(* IEC 61131-3 sources: GHEP-MITSU_BACKUP/, 12 files *)

(* ---- encoder_speed_calc.st ---- *)
(* ============================================================================ *)
(* PROGRAM: POU_ENCODER_SPEED (Fixed Scan 10ms - Ngắt chu kỳ 10ms)             *)
(* MACHINE: MÁY GHÉP MÀNG METALIZE                                             *)
(* HARDWARE: 03 Module QD62 tại Slot 1 (H20), Slot 2 (H30), Slot 3 (H40)        *)
(* ENCODERS: 5 Trục (T = Thu, X1 = Xả 1, X2 = Master, M = Metalize, S = Dầu)     *)
(* ============================================================================ *)

VAR_GLOBAL
    (* --- DỮ LIỆU TỐC ĐỘ ĐỌC VỀ VÀ TÍNH TOÁN (HMI / PROGRAM DÙNG CHUNG) --- *)
    (* Tốc độ vòng/phút (RPM x10: 1500 -> 150.0 RPM) *)
    RPM_T       : DINT := 0; (* Trục Thu T *)
    RPM_X1      : DINT := 0; (* Trục Xả X1 *)
    RPM_X2      : DINT := 0; (* Trục Master X2 *)
    RPM_M       : DINT := 0; (* Trục Metalize M *)
    RPM_S       : DINT := 0; (* Trục Dầu S *)

    (* Tốc độ dây mét/phút (MPM x10: 1205 -> 120.5 MPM) *)
    MPM_T       : DINT := 0; (* Vận tốc dây Trục Thu T *)
    MPM_X1      : DINT := 0; (* Vận tốc dây Trục Xả X1 *)
    MPM_X2      : DINT := 0; (* Vận tốc dây Trục Master X2 (Tốc độ chuẩn dòng máy) *)
    MPM_M       : DINT := 0; (* Vận tốc dây Trục Metalize M *)
    MPM_S       : DINT := 0; (* Vận tốc dây Trục Dầu S *)

    (* Cài đặt đường kính lô (mm) *)
    Dia_T_mm    : DINT := 150; (* Đường kính cuộn Thu T *)
    Dia_X1_mm   : DINT := 150; (* Đường kính cuộn Xả X1 *)
    Dia_X2_mm   : DINT := 200; (* Đường kính lô Master X2 (Cố định 200mm) *)
    Dia_M_mm    : DINT := 180; (* Đường kính lô Metalize M *)
    Dia_S_mm    : DINT := 160; (* Đường kính lô Dầu S *)

    (* Cài đặt độ phân giải Encoder PPR (xung/vòng) *)
    PPR_Encoder : DINT := 2000; (* 2000 PPR x 4 = 8000 pulses/rev *)

    (* Biến lưu xung vòng trước *)
    Prev_Pulse_T  : DINT := 0;
    Prev_Pulse_X1 : DINT := 0;
    Prev_Pulse_X2 : DINT := 0;
    Prev_Pulse_M  : DINT := 0;
    Prev_Pulse_S  : DINT := 0;
END_VAR

VAR
    (* Biến xung hiện tại đọc từ Buffer Memory QD62 *)
    Curr_Pulse_T  : DINT := 0;
    Curr_Pulse_X1 : DINT := 0;
    Curr_Pulse_X2 : DINT := 0;
    Curr_Pulse_M  : DINT := 0;
    Curr_Pulse_S  : DINT := 0;

    (* Delta xung đếm được trong 10ms *)
    Delta_T  : DINT := 0;
    Delta_X1 : DINT := 0;
    Delta_X2 : DINT := 0;
    Delta_M  : DINT := 0;
    Delta_S  : DINT := 0;

    (* PPR tổng sau khi nhân 4 pha A/B *)
    Total_PPR : DINT := 8000;
END_VAR

(* ============================================================================ *)
(* MAIN BODY: CHẠY TRONG POU CHU KỲ NGẮT FIXED SCAN 10MS                      *)
(* ============================================================================ *)

(* --- 1. KÍCH HOẠT CỜ CHO PHÉP ĐẾM XUNG CHO 3 MODULE QD62 --- *)
Y21 := TRUE; (* QD62 #1 (Slot 1 H20) CH1: Enable Trục Thu T *)
Y22 := TRUE; (* QD62 #1 (Slot 1 H20) CH2: Enable Trục Xả X1 *)

Y31 := TRUE; (* QD62 #2 (Slot 2 H30) CH1: Enable Trục Master X2 *)
Y32 := TRUE; (* QD62 #2 (Slot 2 H30) CH2: Enable Trục Metalize M *)

Y41 := TRUE; (* QD62 #3 (Slot 3 H40) CH1: Enable Trục Dầu S *)

(* --- 2. ĐỌC XUNG 32-BIT TỪ BUFFER MEMORY G2/G3 VÀ G10/G11 --- *)
(* QD62 #1 (Slot 1 - H20) *)
DMOV(TRUE, U1\G2,  Curr_Pulse_T);  (* CH1: Trục Thu T *)
DMOV(TRUE, U1\G10, Curr_Pulse_X1); (* CH2: Trục Xả X1 *)

(* QD62 #2 (Slot 2 - H30) *)
DMOV(TRUE, U2\G2,  Curr_Pulse_X2); (* CH1: Trục Master X2 *)
DMOV(TRUE, U2\G10, Curr_Pulse_M);  (* CH2: Trục Metalize M *)

(* QD62 #3 (Slot 3 - H40) *)
DMOV(TRUE, U3\G2,  Curr_Pulse_S);  (* CH1: Trục Dầu S *)

(* --- 3. TÍNH DELTA XUNG NỐI TIẾP TRONG 10MS (100Hz) --- *)
Delta_T  := ABS(Curr_Pulse_T  - Prev_Pulse_T);
Delta_X1 := ABS(Curr_Pulse_X1 - Prev_Pulse_X1);
Delta_X2 := ABS(Curr_Pulse_X2 - Prev_Pulse_X2);
Delta_M  := ABS(Curr_Pulse_M  - Prev_Pulse_M);
Delta_S  := ABS(Curr_Pulse_S  - Prev_Pulse_S);

(* Cập nhật xung vòng trước *)
Prev_Pulse_T  := Curr_Pulse_T;
Prev_Pulse_X1 := Curr_Pulse_X1;
Prev_Pulse_X2 := Curr_Pulse_X2;
Prev_Pulse_M  := Curr_Pulse_M;
Prev_Pulse_S  := Curr_Pulse_S;

Total_PPR := PPR_Encoder * 4; (* Nhân 4 độ phân giải mode 2-Phase 4x *)

(* --- 4. TÍNH TỐC ĐỘ VÒNG/PHÚT RPM (RPM x10: 1500 -> 150.0 RPM) --- *)
(* Công thức: RPM = (Delta_Pulse * 60000ms / 10ms) / Total_PPR *)
IF Total_PPR > 0 THEN
    RPM_T  := (Delta_T  * 600000) / Total_PPR;
    RPM_X1 := (Delta_X1 * 600000) / Total_PPR;
    RPM_X2 := (Delta_X2 * 600000) / Total_PPR;
    RPM_M  := (Delta_M  * 600000) / Total_PPR;
    RPM_S  := (Delta_S  * 600000) / Total_PPR;
END_IF;

(* --- 5. TÍNH VẬN TỐC DÂY MÉT/PHÚT MPM (MPM x10: 1205 -> 120.5 MPM) --- *)
(* Công thức: MPM = (RPM * PI * Dia_mm) / 1000 *)
(* PI x 1000 = 3142 *)
MPM_T  := (RPM_T  * 3142 * Dia_T_mm)  / 1000000;
MPM_X1 := (RPM_X1 * 3142 * Dia_X1_mm) / 1000000;
MPM_X2 := (RPM_X2 * 3142 * Dia_X2_mm) / 1000000; (* Vận tốc Master dây chuyền *)
MPM_M  := (RPM_M  * 3142 * Dia_M_mm)  / 1000000;
MPM_S  := (RPM_S  * 3142 * Dia_S_mm)  / 1000000;

(* ---- metalize_main_program.st ---- *)
(* ============================================================================ *)
(* MAIN PROGRAM: POU_MAIN_METALIZE (BỔ SUNG CHỐNG TRÙNG MÀNG & CHỐNG KHÔ KEO/DẦU S, Ms) *)
(* PLC: Q02UCPU | Base Rack Slot 0..6                                           *)
(* CỜ M130/M131: BẬT/TẮT TORQUE HÃM M & U KHI DỪNG MÁY CHỐNG TRÙNG MÀNG          *)
(* CỜ M132/M133: QUAY BÒ CHẬM TRỤC S & TRỤC Ms KHI DỪNG MÁY CHỐNG KHÔ KEO/DẦU  *)
(* ============================================================================ *)

VAR_GLOBAL
    (* --- BẢNG ĐIỀU KHIỂN HMI WEINTEK --- *)
    HMI_Auto_Mode       : BOOL := TRUE;
    HMI_Reset_Error     : BOOL := FALSE;
    HMI_Start           : BOOL := FALSE;
    HMI_Stop            : BOOL := FALSE;
    HMI_Inc_Hold        : BOOL := FALSE;
    HMI_Dec_Hold        : BOOL := FALSE;
    HMI_PID_Enable      : BOOL := TRUE;

    (* --- CỜ CHỐNG TRÙNG MÀNG KHI DỪNG MÁY (HOLD TORQUE WHEN STOPPED) --- *)
    Hold_Torque_Stop_M  : BOOL := TRUE;  (* ON: Giữ Torque Thắng M khi dừng chống trùng màng *)
    Hold_Torque_Stop_U  : BOOL := TRUE;  (* ON: Giữ Torque Xả U khi dừng chống trùng màng *)

    (* --- CỜ QUAY BÒ CHẬM CHỐNG KHÔ KEO / DẦU CHO TRỤC S & Ms KHI DỪNG MÁY --- *)
    Anti_Dry_Rotate_S   : BOOL := TRUE;  (* ON: Cho Trục Dầu S quay bò chậm khi dừng máy *)
    Anti_Dry_Rotate_Ms  : BOOL := TRUE;  (* ON: Cho Trục Ghép Ms quay bò chậm khi dừng máy *)
    Anti_Dry_Crawl_Speed: DINT := 10;    (* Tốc độ bò chậm chống khô keo (1.0 m/phút) *)

    (* --- LỆNH BEN NÂNG/HẠ CUỘN MÀNG --- *)
    Lift_Up_T           : BOOL := FALSE;
    Lift_Down_T         : BOOL := FALSE;
    Lift_Up_M           : BOOL := FALSE;
    Lift_Down_M         : BOOL := FALSE;
    Lift_Up_U           : BOOL := FALSE;
    Lift_Down_U         : BOOL := FALSE;

    (* --- ĐIỀU KHIỂN 2 PEN ÉP MÀNG QY40 (Y66, Y67) VÀ NÚT BẤM QX40 (X52, X53) --- *)
    Release_Pen_Speed_MPM: DINT := 20;   (* Tốc độ cài đặt nhả 2 pen khi dừng máy (2.0 m/phút) *)
    Pen1_Cmd            : BOOL := FALSE; (* Trạng thái ON/OFF Pen 1 (Y66) *)
    Pen2_Cmd            : BOOL := FALSE; (* Trạng thái ON/OFF Pen 2 (Y67) *)

    (* --- CÀI ĐẶT TORQUE HÃM MIN / MAX --- *)
    Min_Torque_M        : DINT := 400;
    Max_Torque_M        : DINT := 2000;
    Init_Holding_Torque_M : DINT := 800;

    Min_Torque_U        : DINT := 500;
    Max_Torque_U        : DINT := 2500;
    Init_Holding_Torque_U : DINT := 1000;

    (* --- ĐƯỜNG KÍNH LÕI CORE DIA VÀ MAX DIA (MM) --- *)
    Core_Dia_T_mm       : DINT := 76;
    Core_Dia_M_mm       : DINT := 76;
    Core_Dia_U_mm       : DINT := 76;

    Max_Dia_T_mm        : DINT := 1000;
    Max_Dia_M_mm        : DINT := 600;
    Max_Dia_U_mm        : DINT := 800;

    (* --- TỈ LỆ TỐC ĐỘ VÀ BÙ TỐC TRỤC S --- *)
    Speed_Ratio_S       : DINT := 1000;
    Speed_Offset_S      : DINT := 0;

    (* --- TỐC ĐỘ CÀI ĐẶT DÂY CHUYỀN --- *)
    Max_Speed_MPM       : DINT := 1000;
    Min_Speed_MPM       : DINT := 20;
    Current_Line_MPM    : DINT := 0;
    Target_Line_MPM     : DINT := 0;

    (* --- TỶ SỐ TRUYỀN GEAR RATIO --- *)
    Gear_Ratio_T        : DINT := 10100;
    Gear_Ratio_X1       : DINT := 8000;
    Gear_Ratio_X2       : DINT := 8000;
    Gear_Ratio_Ms       : DINT := 10000;
    Gear_Ratio_S        : DINT := 10000;
    Gear_Ratio_U        : DINT := 1000;

    (* --- ĐƯỜNG KÍNH LÔ CƠ CẤU (MM x10) --- *)
    Dia_X1_Roller_mm    : DINT := 3005;
    Dia_X2_Roller_mm    : DINT := 3005;
    Dia_Ms_Roller_mm    : DINT := 2000;
    Dia_S_Roller_mm     : DINT := 1000;

    (* --- ĐƯỜNG KÍNH THỰC TẾ ĐÃ ĐƯỢC LỌC THÔNG THẤP (MM) --- *)
    Real_Dia_T_mm       : DINT := 76;
    Real_Dia_M_mm       : DINT := 600;
    Real_Dia_U_mm       : DINT := 800;

    (* --- ĐỘ DÀY MÀNG (MICRON) --- *)
    Thick_Paper_U_um    : DINT := 60;
    Thick_Metalize_M_um : DINT := 20;

    (* --- MÉT HÀNG ĐÃ GHÉP VÀ MÉT CÀI ĐẶT TỰ DỪNG --- *)
    Set_Target_Length   : DINT := 1000;
    Total_Length_Meters : DINT := 0;
    HMI_Reset_Length    : BOOL := FALSE;
    HMI_Reset_Roll_M    : BOOL := FALSE;
    HMI_Reset_Roll_U    : BOOL := FALSE;
    HMI_Reset_Roll_T    : BOOL := FALSE;

    (* --- LỰC CĂNG SP VÀ CALIB --- *)
    SP_Tension_T        : DINT := 1500;
    SP_Tension_X1       : DINT := 1200;
    SP_Tension_M        : DINT := 1000;
    SP_Tension_U        : DINT := 1000;

    Kp_T : DINT := 150; Ki_T : DINT := 20; Kd_T : DINT := 10;
    Kp_X1: DINT := 120; Ki_X1: DINT := 15; Kd_X1: DINT := 8;
    Kp_M : DINT := 100; Ki_M : DINT := 10; Kd_M : DINT := 5;
    Kp_U : DINT := 100; Ki_U : DINT := 10; Kd_U : DINT := 5;

    Zero_Set_T          : BOOL := FALSE;
    Zero_Set_X1         : BOOL := FALSE;
    Zero_Set_M          : BOOL := FALSE;
    Zero_Set_U          : BOOL := FALSE;

    Calib_Gain_T        : DINT := 1000;
    Calib_Gain_X1       : DINT := 1000;
    Calib_Gain_M        : DINT := 1000;
    Calib_Gain_U        : DINT := 1000;
END_VAR

VAR
    State_Machine       : INT := 0;
    Tension_Stable      : BOOL := FALSE;
    Stable_Timer        : INT := 0;
    Stop_Delay_Timer    : INT := 0;

    Trig_X50            : BOOL := FALSE;
    Trig_X51            : BOOL := FALSE;
    Mem_X50             : BOOL := FALSE;
    Mem_X51             : BOOL := FALSE;

    Trig_X52            : BOOL := FALSE; (* Sườn nút bấm Pen 1 X52 *)
    Mem_X52             : BOOL := FALSE;
    Trig_X53            : BOOL := FALSE; (* Sườn nút bấm Pen 2 X53 *)
    Mem_X53             : BOOL := FALSE;

    Curr_Pulse_X2       : DINT := 0;
    Prev_Pulse_X2       : DINT := 0;
    Accum_Pulse_X2      : DINT := 0;

    Curr_Pulse_T        : DINT := 0;
    Prev_Pulse_T        : DINT := 0;
    Accum_Pulse_T       : DINT := 0;
    Rev_Count_T         : DINT := 0;
    Rev_Count_M         : DINT := 0;
    Rev_Count_U         : DINT := 0;

    (* BIẾN LƯU XUNG ĐỂ TÍNH ĐƯỜNG KÍNH THEO TỶ SỐ XUNG KHI MÁY CHẠY (KHÔNG DÙNG ĐỘ DÀY) *)
    Last_Pulse_X2_M     : DINT := 0;
    Last_Pulse_X2_U     : DINT := 0;
    Last_Pulse_X2_T     : DINT := 0;
    Last_Pulse_T        : DINT := 0;
    Delta_Pulse_M       : DINT := 0;
    Delta_Pulse_U       : DINT := 0;
    Delta_Pulse_T_Master: DINT := 0;

    Raw_Dia_M_mm        : DINT := 600;
    Raw_Dia_U_mm        : DINT := 800;
    Raw_Dia_T_mm        : DINT := 76;

    Calc_Speed_T        : DINT := 0;
    Calc_Speed_X1       : DINT := 0;
    Calc_Speed_X2       : DINT := 0;
    Calc_Speed_Ms       : DINT := 0;
    Calc_Torque_M       : DINT := 0;
    Calc_Speed_S        : DINT := 0;
    Calc_Speed_U        : DINT := 0;

    Base_Torque_M       : DINT := 0;

    pid_T               : FB_TENSION_PID;
    pid_X1              : FB_TENSION_PID;
    pid_M               : FB_TENSION_PID;
    pid_U               : FB_TENSION_PID;

    fbCCLink            : FFB_METALIZE_CONTROL;
END_VAR

(* ============================================================================ *)
(* MAIN LOGIC                                                                   *)
(* ============================================================================ *)

(* 1. ĐIỀU KHIỂN BEN NÂNG / HẠ CUỘN MÀNG T, M, U (QY40P SLOT 5 Y60..Y65) *)
Y60 := Lift_Up_T   AND NOT(Lift_Down_T);
Y61 := Lift_Down_T AND NOT(Lift_Up_T);

Y62 := Lift_Up_M   AND NOT(Lift_Down_M);
Y63 := Lift_Down_M AND NOT(Lift_Up_M);

Y64 := Lift_Up_U   AND NOT(Lift_Down_U);
Y65 := Lift_Down_U AND NOT(Lift_Up_U);

(* 1.1 ĐIỀU KHIỂN 2 PEN ÉP MÀNG QY40 (Y66, Y67) BẰNG 2 NÚT BẤM TOGGLE QX40 (X52, X53) *)
(* Bắt sườn lên sút nhấn X52 (Pen 1) và X53 (Pen 2) trên QX40 *)
Trig_X52 := X52 AND NOT(Mem_X52);
Mem_X52  := X52;

Trig_X53 := X53 AND NOT(Mem_X53);
Mem_X53  := X53;

(* Khi bấm nút X52: Đảo trạng thái Pen 1 (ON -> OFF / OFF -> ON) *)
IF Trig_X52 THEN
    Pen1_Cmd := NOT Pen1_Cmd;
END_IF;

(* Khi bấm nút X53: Đảo trạng thái Pen 2 (ON -> OFF / OFF -> ON) *)
IF Trig_X53 THEN
    Pen2_Cmd := NOT Pen2_Cmd;
END_IF;

(* TỰ ĐỘNG NHẢ 2 PEN KHI MÁY DỪNG ĐẾN TỐC ĐỘ CÀI ĐẶT (Release_Pen_Speed_MPM) *)
(* Khi dừng máy (State 3 Stopping hoặc State 0 Stopped) và tốc độ giảm xuống <= tốc độ cài đặt *)
IF (State_Machine = 3 OR State_Machine = 0) AND (Current_Line_MPM <= Release_Pen_Speed_MPM) THEN
    Pen1_Cmd := FALSE;
    Pen2_Cmd := FALSE;
END_IF;

(* Xuất ngõ ra QY40 *)
Y66 := Pen1_Cmd; (* Ngõ ra Pen 1 trên QY40 *)
Y67 := Pen2_Cmd; (* Ngõ ra Pen 2 trên QY40 *)

(* 2. BẮT SƯỜN LÊN CẢM BIẾN TIỆM CẬN ĐO VÒNG QUAY QX40 *)
Trig_X50 := X50 AND NOT(Mem_X50); (* X50: Cuộn Metalize M *)
Mem_X50  := X50;

Trig_X51 := X51 AND NOT(Mem_X51); (* X51: Cuộn Xả Giấy U *)
Mem_X51  := X51;

(* 3. TÍNH ĐƯỜNG KÍNH THỰC TẾ KHÔNG DÙNG ĐỘ DÀY CHO CUỘN METALIZE M (QX40 X50) *)
IF HMI_Reset_Roll_M THEN
    Rev_Count_M        := 0;
    Raw_Dia_M_mm       := Max_Dia_M_mm;
    Real_Dia_M_mm      := Max_Dia_M_mm;
    Last_Pulse_X2_M    := Curr_Pulse_X2;
    HMI_Reset_Roll_M   := FALSE;
ELSIF Trig_X50 THEN
    Rev_Count_M := Rev_Count_M + 1;
    Delta_Pulse_M := Curr_Pulse_X2 - Last_Pulse_X2_M;
    Last_Pulse_X2_M := Curr_Pulse_X2;

    IF Delta_Pulse_M > 0 THEN
        (* Công thức tỷ số xung Master X2 trong 1 vòng quay cuộn M *)
        Raw_Dia_M_mm := (Delta_Pulse_M * Dia_X2_Roller_mm) / 320000;
        IF Raw_Dia_M_mm < Core_Dia_M_mm THEN Raw_Dia_M_mm := Core_Dia_M_mm; END_IF;
        IF Raw_Dia_M_mm > Max_Dia_M_mm THEN Raw_Dia_M_mm := Max_Dia_M_mm; END_IF;
    END_IF;

    IF Rev_Count_M >= 3 THEN
        Real_Dia_M_mm := Real_Dia_M_mm + ((Raw_Dia_M_mm - Real_Dia_M_mm) / 5);
    ELSE
        Real_Dia_M_mm := Max_Dia_M_mm;
    END_IF;
END_IF;

(* 4. TÍNH ĐƯỜNG KÍNH THỰC TẾ KHÔNG DÙNG ĐỘ DÀY CHO CUỘN XẢ GIẤY U (QX40 X51) *)
IF HMI_Reset_Roll_U THEN
    Rev_Count_U        := 0;
    Raw_Dia_U_mm       := Max_Dia_U_mm;
    Real_Dia_U_mm      := Max_Dia_U_mm;
    Last_Pulse_X2_U    := Curr_Pulse_X2;
    HMI_Reset_Roll_U   := FALSE;
ELSIF Trig_X51 THEN
    Rev_Count_U := Rev_Count_U + 1;
    Delta_Pulse_U := Curr_Pulse_X2 - Last_Pulse_X2_U;
    Last_Pulse_X2_U := Curr_Pulse_X2;

    IF Delta_Pulse_U > 0 THEN
        (* Công thức tỷ số xung Master X2 trong 1 vòng quay cuộn U *)
        Raw_Dia_U_mm := (Delta_Pulse_U * Dia_X2_Roller_mm) / 320000;
        IF Raw_Dia_U_mm < Core_Dia_U_mm THEN Raw_Dia_U_mm := Core_Dia_U_mm; END_IF;
        IF Raw_Dia_U_mm > Max_Dia_U_mm THEN Raw_Dia_U_mm := Max_Dia_U_mm; END_IF;
    END_IF;

    IF Rev_Count_U >= 3 THEN
        Real_Dia_U_mm := Real_Dia_U_mm + ((Raw_Dia_U_mm - Real_Dia_U_mm) / 5);
    ELSE
        Real_Dia_U_mm := Max_Dia_U_mm;
    END_IF;
END_IF;

(* 5. TÍNH ĐƯỜNG KÍNH THỰC TẾ KHÔNG DÙNG ĐỘ DÀY CHO CUỘN THU T (ENCODER THU T / MASTER X2) *)
DMOV(TRUE, U1\G2, Curr_Pulse_T);

IF HMI_Reset_Roll_T THEN
    Accum_Pulse_T    := 0;
    Rev_Count_T      := 0;
    Raw_Dia_T_mm     := Core_Dia_T_mm;
    Real_Dia_T_mm    := Core_Dia_T_mm;
    Last_Pulse_X2_T  := Curr_Pulse_X2;
    Last_Pulse_T     := Curr_Pulse_T;
    HMI_Reset_Roll_T := FALSE;
ELSE
    (* Đếm khi cuộn Thu T quay đủ 1 vòng shaft (8000 ppr x 10.1 gear = 80,800 xung T) *)
    IF (Curr_Pulse_T - Last_Pulse_T) >= ((8000 * Gear_Ratio_T) / 1000) THEN
        Rev_Count_T := Rev_Count_T + 1;
        Delta_Pulse_T_Master := Curr_Pulse_X2 - Last_Pulse_X2_T;
        Last_Pulse_X2_T := Curr_Pulse_X2;
        Last_Pulse_T    := Curr_Pulse_T;

        IF Delta_Pulse_T_Master > 0 THEN
            Raw_Dia_T_mm := (Delta_Pulse_T_Master * Dia_X2_Roller_mm) / 320000;
            IF Raw_Dia_T_mm < Core_Dia_T_mm THEN Raw_Dia_T_mm := Core_Dia_T_mm; END_IF;
            IF Raw_Dia_T_mm > Max_Dia_T_mm THEN Raw_Dia_T_mm := Max_Dia_T_mm; END_IF;
        END_IF;

        IF Rev_Count_T >= 3 THEN
            Real_Dia_T_mm := Real_Dia_T_mm + ((Raw_Dia_T_mm - Real_Dia_T_mm) / 5);
        ELSE
            Real_Dia_T_mm := Core_Dia_T_mm;
        END_IF;
    END_IF;
END_IF;

(* 6. ĐO TỔNG CHIỀU DÀI MÉT HÀNG VÀ TỰ ĐỘNG DỪNG KHI ĐẠT TARGET *)
DMOV(TRUE, U2\G2, Curr_Pulse_X2);

IF HMI_Reset_Length THEN
    Accum_Pulse_X2      := 0;
    Total_Length_Meters := 0;
    HMI_Reset_Length    := FALSE;
ELSE
    IF Curr_Pulse_X2 >= Prev_Pulse_X2 THEN Accum_Pulse_X2 := Accum_Pulse_X2 + (Curr_Pulse_X2 - Prev_Pulse_X2); END_IF;
    Prev_Pulse_X2 := Curr_Pulse_X2;
    Total_Length_Meters := (Accum_Pulse_X2 * 944) / 8000000;
END_IF;

(* 7. STATE MACHINE VẬN HÀNH DÂY CHUYỀN (START / STOP / INC / DEC) *)
CASE State_Machine OF
    0: (* STATE_STOPPED *)
        Current_Line_MPM := 0;
        Target_Line_MPM  := 0;
        Tension_Stable   := FALSE;
        Stable_Timer     := 0;
        Stop_Delay_Timer := 0;

        (* CHẾ ĐỘ XỬ LÝ KHI DỪNG MÁY: CHỐNG TRÙNG MÀNG VÀ CHỐNG KHÔ KEO/DẦU S, Ms *)
        M200 := FALSE; (* Servo OFF Thu T *)
        M201 := FALSE; (* Servo OFF X1 *)
        M202 := FALSE; (* Servo OFF Master X2 *)

        (* BẬT SERVO BÒ CHẬM KHI DỪNG MÁY CHO S VÀ Ms NẾU CỜ M132 / M133 BẬT *)
        M203 := Anti_Dry_Rotate_Ms; (* Servo ON Ms quay bò chậm chống khô keo *)
        M204 := Anti_Dry_Rotate_S;  (* Servo ON S quay bò chậm chống khô dầu *)

        IF HMI_Start THEN
            State_Machine := 1;
            HMI_Start     := FALSE;
        END_IF;

    1: (* STATE_STARTUP_MIN *)
        M200 := TRUE; M201 := TRUE; M202 := TRUE; M203 := TRUE; M204 := TRUE;
        Target_Line_MPM := Min_Speed_MPM;

        IF Current_Line_MPM < Target_Line_MPM THEN Current_Line_MPM := Current_Line_MPM + 2; END_IF;

        Stable_Timer := Stable_Timer + 1;
        IF Stable_Timer >= 200 THEN
            Tension_Stable := TRUE;
            State_Machine  := 2;
        END_IF;

        IF HMI_Stop THEN State_Machine := 3; HMI_Stop := FALSE; END_IF;

    2: (* STATE_RUNNING *)
        M200 := TRUE; M201 := TRUE; M202 := TRUE; M203 := TRUE; M204 := TRUE;

        IF HMI_Inc_Hold THEN
            Target_Line_MPM := Target_Line_MPM + 5;
            IF Target_Line_MPM > Max_Speed_MPM THEN Target_Line_MPM := Max_Speed_MPM; END_IF;
        ELSIF HMI_Dec_Hold THEN
            Target_Line_MPM := Target_Line_MPM - 5;
            IF Target_Line_MPM < Min_Speed_MPM THEN Target_Line_MPM := Min_Speed_MPM; END_IF;
        END_IF;

        IF Current_Line_MPM < Target_Line_MPM THEN Current_Line_MPM := Current_Line_MPM + 3;
        ELSIF Current_Line_MPM > Target_Line_MPM THEN Current_Line_MPM := Current_Line_MPM - 3; END_IF;

        IF (Set_Target_Length > 0 AND Total_Length_Meters >= Set_Target_Length) OR HMI_Stop THEN
            State_Machine := 3;
            HMI_Stop      := FALSE;
        END_IF;

    3: (* STATE_STOPPING *)
        Target_Line_MPM := Min_Speed_MPM;

        IF Current_Line_MPM > Min_Speed_MPM THEN
            Current_Line_MPM := Current_Line_MPM - 4;
            IF Current_Line_MPM < Min_Speed_MPM THEN Current_Line_MPM := Min_Speed_MPM; END_IF;
        ELSE
            Stop_Delay_Timer := Stop_Delay_Timer + 1;
            IF Stop_Delay_Timer >= 200 THEN
                State_Machine := 0;
            END_IF;
        END_IF;
END_CASE;

(* 8. TÍNH BỘ PID LỰC CĂNG CHO T, X1, M (Thắng Từ) VÀ U *)
pid_T(Enable := HMI_PID_Enable, Setpoint := SP_Tension_T, Feedback := fbCCLink.Weight_Net_T, Kp := Kp_T, Ki := Ki_T, Kd := Kd_T);
pid_X1(Enable := HMI_PID_Enable, Setpoint := SP_Tension_X1, Feedback := fbCCLink.Weight_Net_X1, Kp := Kp_X1, Ki := Ki_X1, Kd := Kd_X1);
pid_M(Enable := HMI_PID_Enable, Setpoint := SP_Tension_M, Feedback := fbCCLink.Weight_Net_M, Kp := Kp_M, Ki := Ki_M, Kd := Kd_M);
pid_U(Enable := HMI_PID_Enable, Setpoint := SP_Tension_U, Feedback := fbCCLink.Weight_Net_U, Kp := Kp_U, Ki := Ki_U, Kd := Kd_U);

(* Quy đổi Tốc độ m/phút sang dải 0..4000 DAC *)
Calc_Speed_X2 := (Current_Line_MPM * 4000) / Max_Speed_MPM;

IF State_Machine = 0 THEN
    (* XỬ LÝ TỐC ĐỘ VÀ TORQUE KHI DỪNG MÁY (STATE_MACHINE = 0) *)
    Calc_Speed_T  := 0;
    Calc_Speed_X1 := 0;

    (* BÒ CHẬM TRỤC Ms NẾU BẬT CỜ M133 *)
    IF Anti_Dry_Rotate_Ms THEN
        Calc_Speed_Ms := (Anti_Dry_Crawl_Speed * 4000) / Max_Speed_MPM; (* Chạy bò chậm (1.0 m/p) *)
    ELSE
        Calc_Speed_Ms := 0;
    END_IF;

    (* BÒ CHẬM TRỤC S NẾU BẬT CỜ M132 *)
    IF Anti_Dry_Rotate_S THEN
        Calc_Speed_S := (Anti_Dry_Crawl_Speed * 4000) / Max_Speed_MPM; (* Chạy bò chậm (1.0 m/p) *)
    ELSE
        Calc_Speed_S := 0;
    END_IF;

    (* GIỮ TORQUE HÃM THẮNG M KHI DỪNG CHỐNG TRÙNG MÀNG NẾU BẬT CỜ M130 *)
    IF Hold_Torque_Stop_M THEN
        Calc_Torque_M := Base_Torque_M;
    ELSE
        Calc_Torque_M := 0;
    END_IF;

    (* GIỮ TORQUE XẢ U KHI DỪNG CHỐNG TRÙNG MÀNG NẾU BẬT CỜ M131 *)
    IF Hold_Torque_Stop_U THEN
        Calc_Speed_U := Init_Holding_Torque_U;
    ELSE
        Calc_Speed_U := 0;
    END_IF;
ELSE
    (* CHẠY TỰ ĐỘNG BÌNH THƯỜNG KHI MÁY ĐANG CHẠY *)
    IF Real_Dia_T_mm > 0 THEN Calc_Speed_T := ((Calc_Speed_X2 * Real_Dia_T_mm) / Core_Dia_T_mm) + pid_T.PID_Output; ELSE Calc_Speed_T := Calc_Speed_X2 + pid_T.PID_Output; END_IF;
    Calc_Speed_X1 := Calc_Speed_X2 + pid_X1.PID_Output;
    Calc_Speed_Ms := Calc_Speed_X2;
    Calc_Speed_S  := ((Calc_Speed_X2 * Speed_Ratio_S) / 1000) + Speed_Offset_S;
    IF Real_Dia_U_mm > 0 THEN Calc_Speed_U := ((Calc_Speed_X2 * Max_Dia_U_mm) / Real_Dia_U_mm) + pid_U.PID_Output; ELSE Calc_Speed_U := Calc_Speed_X2 + pid_U.PID_Output; END_IF;

    IF Rev_Count_M < 5 THEN
        Base_Torque_M := Init_Holding_Torque_M;
    ELSE
        IF (Max_Dia_M_mm - Core_Dia_M_mm) > 0 THEN
            Base_Torque_M := Min_Torque_M + (((Real_Dia_M_mm - Core_Dia_M_mm) * (Max_Torque_M - Min_Torque_M)) / (Max_Dia_M_mm - Core_Dia_M_mm));
        ELSE
            Base_Torque_M := Min_Torque_M;
        END_IF;
    END_IF;

    Calc_Torque_M := Base_Torque_M + pid_M.PID_Output;
END_IF;

(* Ép biên an toàn *)
IF Calc_Speed_T  < 0 THEN Calc_Speed_T  := 0; ELSIF Calc_Speed_T  > 4000 THEN Calc_Speed_T  := 4000; END_IF;
IF Calc_Speed_X1 < 0 THEN Calc_Speed_X1 := 0; ELSIF Calc_Speed_X1 > 4000 THEN Calc_Speed_X1 := 4000; END_IF;
IF Calc_Speed_Ms < 0 THEN Calc_Speed_Ms := 0; ELSIF Calc_Speed_Ms > 4000 THEN Calc_Speed_Ms := 4000; END_IF;
IF Calc_Torque_M < 0 THEN Calc_Torque_M := 0; ELSIF Calc_Torque_M > 4000 THEN Calc_Torque_M := 4000; END_IF;
IF Calc_Speed_S  < 0 THEN Calc_Speed_S  := 0; ELSIF Calc_Speed_S  > 4000 THEN Calc_Speed_S  := 4000; END_IF;
IF Calc_Speed_U  < 0 THEN Calc_Speed_U  := 0; ELSIF Calc_Speed_U  > 4000 THEN Calc_Speed_U  := 4000; END_IF;

D600 := INT_TO_WORD(Calc_Speed_T);
D601 := INT_TO_WORD(pid_T.PID_Output);
D602 := INT_TO_WORD(Calc_Speed_X1);
D603 := INT_TO_WORD(Calc_Speed_X2);
D604 := INT_TO_WORD(Calc_Speed_Ms);
D605 := INT_TO_WORD(Calc_Torque_M);
D606 := INT_TO_WORD(Calc_Speed_S);
D607 := INT_TO_WORD(Calc_Speed_U);

fbCCLink(
    Enable          := TRUE,
    ResetErr        := HMI_Reset_Error,
    Auto_Mode       := HMI_Auto_Mode,

    Zero_Set_T      := Zero_Set_T,
    Zero_Set_X1     := Zero_Set_X1,
    Zero_Set_M      := Zero_Set_M,
    Zero_Set_U      := Zero_Set_U,

    Calib_Gain_T    := Calib_Gain_T,
    Calib_Gain_X1   := Calib_Gain_X1,
    Calib_Gain_M    := Calib_Gain_M,
    Calib_Gain_U    := Calib_Gain_U,

    Set_Speed_T     := D600,
    Set_Torque_T    := D601,
    Set_Speed_X1    := D602,
    Set_Speed_X2    := D603,
    Set_Speed_Ms    := D604,
    Set_Torque_M    := D605,
    Set_Speed_S     := D606,
    Set_Speed_U     := D607,

    Auto_Son_T      := M200,
    Auto_Son_X1     := M201,
    Auto_Son_X2     := M202,
    Auto_Son_M      := M203,
    Auto_Son_S      := M204,

    Test_Son_T      := M210,
    Test_Son_X1     := M211,
    Test_Son_X2     := M212,
    Test_Son_M      := M213,
    Test_Son_S      := M214,

    Test_Speed_T    := D610,
    Test_Speed_X1   := D611,
    Test_Speed_X2   := D612,
    Test_Speed_Ms   := D613,
    Test_Torque_M   := D614,
    Test_Speed_S    := D615,
    Test_Speed_U    := D616
);

(* ---- metalize_pid_control.st ---- *)
(* ============================================================================ *)
(* FUNCTION BLOCK: FB_TENSION_PID (THUẬT TOÁN PID LỰC CĂNG CHUYÊN DỤNG MÁY GHÉP)  *)
(* TÍCH HỢP: ANTI-WINDUP, DEADBAND (VÙNG CHẾT), HẠN CHẾ VỌNG TỐC VÀ ÉP BIÊN    *)
(* ============================================================================ *)

FUNCTION_BLOCK FB_TENSION_PID
VAR_INPUT
    Enable          : BOOL := TRUE;  (* Bật PID *)
    Reset           : BOOL := FALSE; (* Reset tích lũy I *)

    Setpoint        : DINT := 1000;  (* Giá trị lực căng cài đặt (N hoặc Kg) *)
    Feedback        : DINT := 1000;  (* Tải trọng phản hồi từ Loadcell Net *)

    Kp              : DINT := 100;   (* Hệ số P (x100: 100 = 1.00) *)
    Ki              : DINT := 10;    (* Hệ số I (x100: 10 = 0.10) *)
    Kd              : DINT := 5;     (* Hệ số D (x100: 5 = 0.05) *)

    Deadband        : DINT := 10;    (* Vùng chết không chỉnh (N/Kg) *)
    Out_Min         : DINT := -1000; (* Giới hạn đầu ra tối thiểu *)
    Out_Max         : DINT := 1000;  (* Giới hạn đầu ra tối đa *)
END_VAR

VAR_OUTPUT
    PID_Output      : DINT := 0;     (* Giá trị bù tốc độ/torque cho DAC *)
    Error           : DINT := 0;     (* Độ lệch e(k) *)
END_VAR

VAR
    Error_Prev      : DINT := 0;
    I_Term          : DINT := 0;
    P_Term          : DINT := 0;
    D_Term          : DINT := 0;
END_VAR

IF NOT Enable THEN
    PID_Output := 0;
    I_Term     := 0;
    Error_Prev := 0;
    RETURN;
END_IF;

IF Reset THEN
    I_Term     := 0;
    Error_Prev := 0;
    PID_Output := 0;
    RETURN;
END_IF;

(* 1. TÍNH ĐỘ LỆCH ERROR E(K) *)
Error := Setpoint - Feedback;

(* 2. BỘ LỌC VÙNG CHẾT DEADBAND *)
IF ABS(Error) <= Deadband THEN
    Error := 0;
END_IF;

(* 3. TÍNH THÀNH PHẦN PROPORTIONAL (P) *)
P_Term := (Error * Kp) / 100;

(* 4. TÍNH THÀNH PHẦN INTEGRAL (I) VỚI CHỐNG BÃO HÒA ANTI-WINDUP *)
I_Term := I_Term + ((Error * Ki) / 100);

IF I_Term > Out_Max THEN
    I_Term := Out_Max;
ELSIF I_Term < Out_Min THEN
    I_Term := Out_Min;
END_IF;

(* 5. TÍNH THÀNH PHẦN DERIVATIVE (D) *)
D_Term := ((Error - Error_Prev) * Kd) / 100;
Error_Prev := Error;

(* 6. TỔNG HỢP NỔI PID VÀ ÉP BIÊN OUT_MIN..OUT_MAX *)
PID_Output := P_Term + I_Term + D_Term;

IF PID_Output > Out_Max THEN
    PID_Output := Out_Max;
ELSIF PID_Output < Out_Min THEN
    PID_Output := Out_Min;
END_IF;

END_FUNCTION_BLOCK

(* ---- cclink_control.st ---- *)
(* ============================================================================ *)
(* PROGRAM: POU_CCLINK_CONTROL                                                  *)
(* HARDWARE: PLC Q02UCPU + Master QJ61BT11N (Slot 0)                             *)
(* BASE ADDRESSES: Remote Input (RX) = M1008 | Remote Output (RY) = M1200        *)
(* ============================================================================ *)

(* --- 1. CC-LINK NETWORK MONITOR & HANDSHAKE INITIALIZATION --- *)
(* Cờ SB0020 = TRUE: Mạng truyền thông CC-Link hoạt động bình thường *)
IF SB0020 THEN

    (* Kích hoạt cho phép chuyển đổi A/D kênh 1..4 trên AJ65SBT-64AD (Trạm 1) *)
    M1208 := TRUE;  (* RY8: AD Conversion Enable (M1200 + 8) *)

    (* Kích hoạt cho phép xuất Analog D/A kênh 1..8 trên AJ65VBTCU-68DAVN (Trạm 2) *)
    M1240 := TRUE;  (* RY28: DA Conversion Enable (M1200 + 40) *)

ELSE
    (* Trường hợp truyền thông CC-Link bị lỗi *)
    M1208 := FALSE;
    M1240 := FALSE;
END_IF;

(* --- 2. ĐỌC VÀ QUY ĐỔI DỮ LIỆU ANALOG INPUT (AJ65SBT-64AD) --- *)
(* RWr0..RWr3 tự động map về D500..D503 *)
(* D500: Raw CH1 (0..4000) -> Quy đổi sang % D600 (0..1000 = 0.0%..100.0%) *)
IF M1016 THEN (* RX8: AD Conversion Completion Flag (M1008 + 8) *)

    (* Kênh CH1 Analog Input *)
    D600 := INT_TO_WORD(WORD_TO_INT(D500) * 1000 / 4000);

    (* Kênh CH2 Analog Input *)
    D601 := INT_TO_WORD(WORD_TO_INT(D501) * 1000 / 4000);

    (* Kênh CH3 Analog Input *)
    D602 := INT_TO_WORD(WORD_TO_INT(D502) * 1000 / 4000);

    (* Kênh CH4 Analog Input *)
    D603 := INT_TO_WORD(WORD_TO_INT(D503) * 1000 / 4000);

END_IF;

(* --- 3. XUẤT DỮ LIỆU ANALOG OUTPUT (AJ65VBTCU-68DAVN) --- *)
(* D610..D617 chứa giá trị cài đặt (0..1000 = 0.0%..100.0%) *)
(* Quy đổi sang dải DAC (-4000..+4000 hoặc 0..4000) để ghi vào RWw4..RWwB (D524..D531) *)

(* CH1 Analog Output Command *)
D524 := INT_TO_WORD(WORD_TO_INT(D610) * 4000 / 1000);

(* CH2 Analog Output Command *)
D525 := INT_TO_WORD(WORD_TO_INT(D611) * 4000 / 1000);

(* CH3 Analog Output Command *)
D526 := INT_TO_WORD(WORD_TO_INT(D612) * 4000 / 1000);

(* CH4 Analog Output Command *)
D527 := INT_TO_WORD(WORD_TO_INT(D613) * 4000 / 1000);

(* CH5 Analog Output Command *)
D528 := INT_TO_WORD(WORD_TO_INT(D614) * 4000 / 1000);

(* CH6 Analog Output Command *)
D529 := INT_TO_WORD(WORD_TO_INT(D615) * 4000 / 1000);

(* CH7 Analog Output Command *)
D530 := INT_TO_WORD(WORD_TO_INT(D616) * 4000 / 1000);

(* CH8 Analog Output Command *)
D531 := INT_TO_WORD(WORD_TO_INT(D617) * 4000 / 1000);

(* --- 4. ĐIỀU KHIỂN REMOTE DIGITAL I/O (AJ65SBT-16DT - TRẠM 4) --- *)
(* Đọc 8 bit Remote Input M1104..M1111 *)
(* Ghi 8 bit Remote Output M1296..M1303 *)

(* Bật ngõ ra Y0 (M1296) khi nút nhấn X0 (M1104) được ấn và truyền thông OK *)
M1296 := M1104 AND SB0020;

(* Bật ngõ ra Y1 (M1297) theo trạng thái nút nhấn X1 (M1105) *)
M1297 := M1105 AND SB0020;

(* Bật đèn báo lỗi (M1303 - Y7) nếu CC-Link có lỗi hoặc module báo lỗi *)
M1303 := NOT(SB0020) OR M1032 OR M1066;

(* --- 5. RESET LỖI KHI BẤM NÚT RESET (M1111 - X7) --- *)
IF M1111 THEN
    M1226 := TRUE; (* RY1A: Reset lỗi AJ65SBT-64AD *)
    M1258 := TRUE; (* RY3A: Reset lỗi AJ65VBTCU-68DAVN *)
ELSE
    M1226 := FALSE;
    M1258 := FALSE;
END_IF;

(* ---- fb_cclink_control.st ---- *)
(******************************************************************************)
(* PHẦN 1: KHAI BÁO CÁC NHÃN TRONG CỬA SỔ LOCAL LABEL CỦA FB                 *)
(******************************************************************************)
(*
--- BẢNG VAR_INPUT (Class: VAR_INPUT) ---
Label Name      Data Type   Initial Value   Comment
Enable          BOOL        TRUE            Cho phép khối FB hoạt động
ResetErr        BOOL        FALSE           Nút reset lỗi hệ thống
DAC_CH1_Set     WORD        0               Cài đặt DAC CH1 (0..1000 = 0..100.0%)
DAC_CH2_Set     WORD        0               Cài đặt DAC CH2 (0..1000 = 0..100.0%)
DAC_CH3_Set     WORD        0               Cài đặt DAC CH3 (0..1000 = 0..100.0%)
DAC_CH4_Set     WORD        0               Cài đặt DAC CH4 (0..1000 = 0..100.0%)
DAC_CH5_Set     WORD        0               Cài đặt DAC CH5 (0..1000 = 0..100.0%)
DAC_CH6_Set     WORD        0               Cài đặt DAC CH6 (0..1000 = 0..100.0%)
DAC_CH7_Set     WORD        0               Cài đặt DAC CH7 (0..1000 = 0..100.0%)
DAC_CH8_Set     WORD        0               Cài đặt DAC CH8 (0..1000 = 0..100.0%)
DO_Y0_Cmd       BOOL        FALSE           Lệnh ngõ ra Y0 St 4 (M1296)
DO_Y1_Cmd       BOOL        FALSE           Lệnh ngõ ra Y1 St 4 (M1297)

--- BẢNG VAR_OUTPUT (Class: VAR_OUTPUT) ---
Label Name      Data Type   Initial Value   Comment
CCLink_OK       BOOL        FALSE           Trạng thái mạng CC-Link OK
HasError        BOOL        FALSE           Báo lỗi tổng truyền thông/module
ADC_CH1_Val     WORD        0               Giá trị % ADC CH1 (0..1000)
ADC_CH2_Val     WORD        0               Giá trị % ADC CH2 (0..1000)
ADC_CH3_Val     WORD        0               Giá trị % ADC CH3 (0..1000)
ADC_CH4_Val     WORD        0               Giá trị % ADC CH4 (0..1000)
ADC_CH1_Raw     WORD        0               Giá trị thô D500 ADC CH1 (0..4000)
ADC_CH2_Raw     WORD        0               Giá trị thô D501 ADC CH2 (0..4000)
ADC_CH3_Raw     WORD        0               Giá trị thô D502 ADC CH3 (0..4000)
ADC_CH4_Raw     WORD        0               Giá trị thô D503 ADC CH4 (0..4000)
DI_X0_State     BOOL        FALSE           Trạng thái ngõ vào X0 St 4 (M1104)
DI_X1_State     BOOL        FALSE           Trạng thái ngõ vào X1 St 4 (M1105)
*)

(******************************************************************************)
(* PHẦN 2: MÃ ST CHÍNH (COPY DÁN VÀO KHUNG CHƯƠNG TRÌNH ST CỦA FB)            *)
(******************************************************************************)

IF Enable THEN

    (* 1. Kiểm tra trạng thái mạng CC-Link & Ghi 1 lần tránh cảnh báo C9300 *)
    CCLink_OK := SB0020;
    HasError  := NOT(SB0020) OR M1032 OR M1066;

    M1208 := SB0020;  (* RY8: AD Conversion Enable *)
    M1240 := SB0020;  (* RY28: DA Conversion Enable *)

    (* 2. Đọc 4 kênh Analog Input (AJ65SBT-64AD) *)
    IF M1016 THEN (* RX8: AD Conversion Completed *)
        ADC_CH1_Raw := D500;
        ADC_CH2_Raw := D501;
        ADC_CH3_Raw := D502;
        ADC_CH4_Raw := D503;

        (* Quy đổi sang 0..1000 (0.0% .. 100.0%) *)
        ADC_CH1_Val := INT_TO_WORD(WORD_TO_INT(D500) * 1000 / 4000);
        ADC_CH2_Val := INT_TO_WORD(WORD_TO_INT(D501) * 1000 / 4000);
        ADC_CH3_Val := INT_TO_WORD(WORD_TO_INT(D502) * 1000 / 4000);
        ADC_CH4_Val := INT_TO_WORD(WORD_TO_INT(D503) * 1000 / 4000);
    END_IF;

    (* 3. Ghi 8 kênh Analog Output (AJ65VBTCU-68DAVN) *)
    D524 := INT_TO_WORD(WORD_TO_INT(DAC_CH1_Set) * 4000 / 1000);
    D525 := INT_TO_WORD(WORD_TO_INT(DAC_CH2_Set) * 4000 / 1000);
    D526 := INT_TO_WORD(WORD_TO_INT(DAC_CH3_Set) * 4000 / 1000);
    D527 := INT_TO_WORD(WORD_TO_INT(DAC_CH4_Set) * 4000 / 1000);
    D528 := INT_TO_WORD(WORD_TO_INT(DAC_CH5_Set) * 4000 / 1000);
    D529 := INT_TO_WORD(WORD_TO_INT(DAC_CH6_Set) * 4000 / 1000);
    D530 := INT_TO_WORD(WORD_TO_INT(DAC_CH7_Set) * 4000 / 1000);
    D531 := INT_TO_WORD(WORD_TO_INT(DAC_CH8_Set) * 4000 / 1000);

    (* 4. Xử lý Digital Remote I/O (AJ65SBT-16DT) *)
    DI_X0_State := M1104;
    DI_X1_State := M1105;

    M1296 := DO_Y0_Cmd AND SB0020;
    M1297 := DO_Y1_Cmd AND SB0020;
    M1303 := HasError;

    (* 5. Reset lỗi (Ghi 1 lần tránh cảnh báo C9300) *)
    M1226 := ResetErr OR M1111; (* RY1A: Reset lỗi AJ65SBT-64AD *)
    M1258 := ResetErr OR M1111; (* RY3A: Reset lỗi AJ65VBTCU-68DAVN *)

END_IF;

(* ---- fb_code_body.st ---- *)
IF Enable THEN

    (* 1. Kiem tra trang thai mang CC-Link & Ghi 1 lan duy nhat (Tranh canh bao C9300) *)
    CCLink_OK := SB0020;
    HasError  := NOT(SB0020) OR M1032 OR M1066;

    M1208 := SB0020;  (* RY8: AD Conversion Enable (St 1) *)
    M1240 := SB0020;  (* RY28: DA Conversion Enable (St 2) *)

    (* 2. Doc 4 kenh Analog Input (AJ65SBT-64AD - Tram 1) *)
    IF M1016 THEN (* RX8: AD Conversion Completed *)
        ADC_CH1_Raw := D500;
        ADC_CH2_Raw := D501;
        ADC_CH3_Raw := D502;
        ADC_CH4_Raw := D503;

        (* Quy doi sang 0..1000 (0.0% .. 100.0%) *)
        ADC_CH1_Val := INT_TO_WORD(WORD_TO_INT(D500) * 1000 / 4000);
        ADC_CH2_Val := INT_TO_WORD(WORD_TO_INT(D501) * 1000 / 4000);
        ADC_CH3_Val := INT_TO_WORD(WORD_TO_INT(D502) * 1000 / 4000);
        ADC_CH4_Val := INT_TO_WORD(WORD_TO_INT(D503) * 1000 / 4000);
    END_IF;

    (* 3. Ghi 8 kenh Analog Output (AJ65VBTCU-68DAVN - Tram 2 & 3) *)
    (* QUY ĐỔI LỆNH 0..4000 XUẤT RA ĐIỆN ÁP THỰC TẾ 0..5V *)
    (* (Vi dải dac 0..10V tuong ung 0..4000, nen de xuat 0..5V ta lay User_Cmd / 2) *)
    D524 := INT_TO_WORD(WORD_TO_INT(DAC_CH1_Set) / 2); (* CH1 Output 0..5V *)
    D525 := INT_TO_WORD(WORD_TO_INT(DAC_CH2_Set) / 2); (* CH2 Output 0..5V *)
    D526 := INT_TO_WORD(WORD_TO_INT(DAC_CH3_Set) / 2); (* CH3 Output 0..5V *)
    D527 := INT_TO_WORD(WORD_TO_INT(DAC_CH4_Set) / 2); (* CH4 Output 0..5V *)
    D528 := INT_TO_WORD(WORD_TO_INT(DAC_CH5_Set) / 2); (* CH5 Output 0..5V *)
    D529 := INT_TO_WORD(WORD_TO_INT(DAC_CH6_Set) / 2); (* CH6 Output 0..5V *)
    D530 := INT_TO_WORD(WORD_TO_INT(DAC_CH7_Set) / 2); (* CH7 Output 0..5V *)
    D531 := INT_TO_WORD(WORD_TO_INT(DAC_CH8_Set) / 2); (* CH8 Output 0..5V *)

    (* 4. Xu ly Digital Remote I/O (AJ65SBT-16DT - Tram 4) *)
    DI_X0_State := M1104;  (* RX60 St 4 *)
    DI_X1_State := M1105;  (* RX61 St 4 *)

    M1296 := DO_Y0_Cmd AND SB0020;  (* RY60 St 4 *)
    M1297 := DO_Y1_Cmd AND SB0020;  (* RY61 St 4 *)
    M1303 := HasError;             (* RY67 St 4 *)

    (* 5. Reset loi *)
    M1226 := ResetErr OR M1111; (* RY1A: Reset loi St 1 *)
    M1258 := ResetErr OR M1111; (* RY3A: Reset loi St 2 *)

END_IF;

(* ---- fb_tension_pid_body.st ---- *)
IF NOT Enable THEN
    PID_Output := 0;
    I_Term     := 0;
    Error_Prev := 0;
    RETURN;
END_IF;

IF Reset THEN
    I_Term     := 0;
    Error_Prev := 0;
    PID_Output := 0;
    RETURN;
END_IF;

(* 1. TÍNH ĐỘ LỆCH ERROR E(K) *)
Error := Setpoint - Feedback;

(* 2. BỘ LỌC VÙNG CHẾT DEADBAND *)
IF ABS(Error) <= Deadband THEN
    Error := 0;
END_IF;

(* 3. TÍNH THÀNH PHẦN PROPORTIONAL (P) *)
P_Term := (Error * Kp) / 100;

(* 4. TÍNH THÀNH PHẦN INTEGRAL (I) VỚI CHỐNG BÃO HÒA ANTI-WINDUP *)
I_Term := I_Term + ((Error * Ki) / 100);

IF I_Term > Out_Max THEN
    I_Term := Out_Max;
ELSIF I_Term < Out_Min THEN
    I_Term := Out_Min;
END_IF;

(* 5. TÍNH THÀNH PHẦN DERIVATIVE (D) *)
D_Term := ((Error - Error_Prev) * Kd) / 100;
Error_Prev := Error;

(* 6. TỔNG HỢP NỔI PID VÀ ÉP BIÊN OUT_MIN..OUT_MAX *)
PID_Output := P_Term + I_Term + D_Term;

IF PID_Output > Out_Max THEN
    PID_Output := Out_Max;
ELSIF PID_Output < Out_Min THEN
    PID_Output := Out_Min;
END_IF;

(* ---- init_program.st ---- *)
(* ============================================================================ *)
(* TÊN CHƯƠNG TRÌNH : INIT_PROGRAM (INITIAL EXECUTION POU - KHỞI TẠO HỆ THỐNG)    *)
(* HỆ THỐNG        : MÁY GHÉP MÀNG METALIZE TỰ ĐỘNG - MITSUBISHI Q02U PLC       *)
(* KIỂU DỮ LIỆU    : SỐ THỰC FLOAT / REAL (CHUẨN IEC)                          *)
(* CẤU TRÚC PHẦN CỨNG MỚI (DIRECT BASE RACK - KHÔNG DÙNG CC-LINK):             *)
(*   - SLOT 0 (H00): Q68ADV (8 CH Analog Input: Loadcell T, X1, M, U & Analog S)*)
(*   - SLOT 1 (H10): Q68DAV (8 CH Analog Output: Speed/Torque T, X1, X2, Ms, S, M, U) *)
(*   - SLOT 2 (H20): QD62D  (2 CH High Speed Counter: Trục T & Trục X1)        *)
(*   - SLOT 3 (H30): QD62D  (2 CH High Speed Counter: Trục X2 & Trục Ms)       *)
(*   - SLOT 4 (H40): QX40   (16 CH Digital Input: X40..X4F)                    *)
(*   - SLOT 5 (H50): QY40   (16 CH Digital Output: Y50..Y5F)                   *)
(*   - SLOT 6 (H60): QJ71C24N (RS232/RS485 Communication)                      *)
(* ============================================================================ *)

(* ---------------------------------------------------------------------------- *)
(* 1. KHỞI TẠO TỐC ĐỘ TỐI ĐA MOTOR (RPM - REAL)                                *)
(* ---------------------------------------------------------------------------- *)
IF Max_RPM_X2 <= 0.0 THEN Max_RPM_X2 := 1000.0; END_IF; (* Trục Master X2: Max 1000 RPM *)
IF Max_RPM_X1 <= 0.0 THEN Max_RPM_X1 := 1000.0; END_IF; (* Trục Kéo X1:    Max 1000 RPM *)
IF Max_RPM_Ms <= 0.0 THEN Max_RPM_Ms := 3000.0; END_IF; (* Trục Ghép Ms:   Max 3000 RPM *)
IF Max_RPM_S  <= 0.0 THEN Max_RPM_S  := 3000.0; END_IF; (* Trục Dầu S:     Max 3000 RPM *)
IF Max_RPM_T  <= 0.0 THEN Max_RPM_T  := 1500.0; END_IF; (* Trục Thu T:     Max 1500 RPM *)

(* ---------------------------------------------------------------------------- *)
(* 2. KHỞI TẠO TỶ SỐ TRUYỀN HỘP SỐ THỰC TẾ (GEAR RATIO - REAL)                *)
(* ---------------------------------------------------------------------------- *)
IF Gear_Ratio_T  <= 0.0 THEN Gear_Ratio_T  := 10.1; END_IF; (* Thu T:     10.1 : 1 (D620) *)
IF Gear_Ratio_X1 <= 0.0 THEN Gear_Ratio_X1 := 8.0;  END_IF; (* Xả X1:     8.0  : 1 (D622) *)
IF Gear_Ratio_X2 <= 0.0 THEN Gear_Ratio_X2 := 8.0;  END_IF; (* Master X2: 8.0  : 1 (D624) *)
IF Gear_Ratio_Ms <= 0.0 THEN Gear_Ratio_Ms := 10.0; END_IF; (* Ghép Ms:   10.0 : 1 (D626) *)
IF Gear_Ratio_S  <= 0.0 THEN Gear_Ratio_S  := 10.0; END_IF; (* Dầu S:     10.0 : 1 (D628) *)
IF Gear_Ratio_U  <= 0.0 THEN Gear_Ratio_U  := 1.0;  END_IF; (* Xả U:      1.0  : 1 (D630) *)

(* ---------------------------------------------------------------------------- *)
(* 3. KHỞI TẠO ĐƯỜNG KÍNH LÔ CƠ CẤU (ROLLER DIAMETER - mm - REAL)              *)
(* ---------------------------------------------------------------------------- *)
IF Dia_X1_Roller_mm <= 0.0 THEN Dia_X1_Roller_mm := 300.5; END_IF; (* Lô Kéo X1:    300.5 mm (D638) *)
IF Dia_X2_Roller_mm <= 0.0 THEN Dia_X2_Roller_mm := 300.5; END_IF; (* Lô Master X2: 300.5 mm (D642) *)
IF Dia_Ms_Roller_mm <= 0.0 THEN Dia_Ms_Roller_mm := 200.0; END_IF; (* Lô Ghép Ms:   200.0 mm (D640) *)
IF Dia_S_Roller_mm  <= 0.0 THEN Dia_S_Roller_mm  := 100.0; END_IF; (* Lô Dầu S:     100.0 mm (D648) *)

(* ---------------------------------------------------------------------------- *)
(* 4. KHỞI TẠO ĐƯỜNG KÍNH LÕI (CORE) VÀ ĐƯỜNG KÍNH MAX (MAX DIA) (mm - REAL)    *)
(* ---------------------------------------------------------------------------- *)
IF Core_Dia_T_mm <= 0.0 THEN Core_Dia_T_mm := 76.0;   END_IF; (* Lõi cuộn Thu T:  76.0 mm (D644) *)
IF Core_Dia_M_mm <= 0.0 THEN Core_Dia_M_mm := 76.0;   END_IF; (* Lõi cuộn Xả M:   76.0 mm (D645) *)
IF Core_Dia_U_mm <= 0.0 THEN Core_Dia_U_mm := 76.0;   END_IF; (* Lõi cuộn Xả U:   76.0 mm (D647) *)

IF Max_Dia_T_mm  <= 0.0 THEN Max_Dia_T_mm  := 1000.0; END_IF; (* Cuộn Thu T max: 1000.0 mm (D646) *)
IF Max_Dia_M_mm  <= 0.0 THEN Max_Dia_M_mm  := 600.0;  END_IF; (* Cuộn Xả M max:   600.0 mm (D649) *)
IF Max_Dia_U_mm  <= 0.0 THEN Max_Dia_U_mm  := 800.0;  END_IF; (* Cuộn Xả U max:   800.0 mm (D650) *)

(* ---------------------------------------------------------------------------- *)
(* 5. KHỞI TẠO ĐƯỜNG KÍNH BAN ĐẦU KHI MỚI BẬT NGUỒN (REAL)                     *)
(* ---------------------------------------------------------------------------- *)
IF Real_Dia_T_mm < Core_Dia_T_mm OR Real_Dia_T_mm > Max_Dia_T_mm THEN
    Real_Dia_T_mm := Core_Dia_T_mm; (* 76.0 mm - D724 *)
END_IF;

IF Real_Dia_M_mm < Core_Dia_M_mm OR Real_Dia_M_mm > Max_Dia_M_mm THEN
    Real_Dia_M_mm := Max_Dia_M_mm;  (* 600.0 mm - D722 *)
END_IF;

IF Real_Dia_U_mm < Core_Dia_U_mm OR Real_Dia_U_mm > Max_Dia_U_mm THEN
    Real_Dia_U_mm := Max_Dia_U_mm;  (* 800.0 mm - D720 *)
END_IF;

(* ---------------------------------------------------------------------------- *)
(* 6. KHỞI TẠO TỶ LỆ TỐC ĐỘ VÀ BÙ TỐC (SPEED RATIO - REAL, 1.0 = 100%)         *)
(* ---------------------------------------------------------------------------- *)
IF Speed_Ratio_T  <= 0.0 THEN Speed_Ratio_T  := 1.05; END_IF; (* Chạy nhanh hơn 5% giữ căng (D756) *)
IF Speed_Ratio_X1 <= 0.0 THEN Speed_Ratio_X1 := 1.00; END_IF; (* Đồng bộ 100.0% (D758) *)
IF Speed_Ratio_Ms <= 0.0 THEN Speed_Ratio_Ms := 1.00; END_IF; (* Đồng bộ 100.0% (D762) *)
IF Speed_Ratio_S  <= 0.0 THEN Speed_Ratio_S  := 1.00; END_IF; (* Đồng bộ 100.0% (D766) *)

(* ---------------------------------------------------------------------------- *)
(* 7. KHỞI TẠO GIỚI HẠN TỐC ĐỘ DÂY CHUYỀN (m/phút - REAL)                      *)
(* ---------------------------------------------------------------------------- *)
IF Max_Speed_MPM         <= 0.0 THEN Max_Speed_MPM         := 100.0; END_IF; (* Max 100.0 m/p (D602) *)
IF Min_Speed_MPM         <= 0.0 THEN Min_Speed_MPM         := 2.0;   END_IF; (* Min 2.0 m/p (D603) *)
IF Release_Pen_Speed_MPM <= 0.0 THEN Release_Pen_Speed_MPM := 2.0;   END_IF; (* Tốc độ nhả pen (D604) *)
IF Ramp_Accel_Rate       <= 0.0 THEN Ramp_Accel_Rate       := 0.5;   END_IF; (* Gia tốc tăng tốc (D606) *)
IF Ramp_Decel_Rate       <= 0.0 THEN Ramp_Decel_Rate       := 1.0;   END_IF; (* Gia tốc giảm tốc (D608) *)
IF Decel_Distance_Meters <= 0.0 THEN Decel_Distance_Meters := 50.0;  END_IF; (* Khoảng cách hãm dừng (m) *)

(* ---------------------------------------------------------------------------- *)
(* 8. KHỞI TẠO CÀI ĐẶT LỰC CĂNG (TENSION SP - kg/N - REAL) & HỆ SỐ PID         *)
(* ---------------------------------------------------------------------------- *)
IF SP_Tension_T  <= 0.0 THEN SP_Tension_T  := 15.0; END_IF; (* SP Lực căng Thu T: 15.0 kg (D660) *)
IF SP_Tension_X1 <= 0.0 THEN SP_Tension_X1 := 12.0; END_IF; (* SP Lực căng Xả X1: 12.0 kg (D662) *)
IF SP_Tension_M  <= 0.0 THEN SP_Tension_M  := 10.0; END_IF; (* SP Lực căng Xả M:  10.0 kg (D664) *)
IF SP_Tension_U  <= 0.0 THEN SP_Tension_U  := 10.0; END_IF; (* SP Lực căng Xả U:  10.0 kg (D668) *)

(* Hệ số PID cuộn Thu T *)
IF Kp_T <= 0.0 THEN Kp_T := 1.5; END_IF;
IF Ki_T <= 0.0 THEN Ki_T := 0.2; END_IF;
IF Kd_T <= 0.0 THEN Kd_T := 0.1; END_IF;

(* Hệ số PID cuộn Xả X1 *)
IF Kp_X1 <= 0.0 THEN Kp_X1 := 1.2; END_IF;
IF Ki_X1 <= 0.0 THEN Ki_X1 := 0.15; END_IF;
IF Kd_X1 <= 0.0 THEN Kd_X1 := 0.08; END_IF;

(* Hệ số PID trục Master X2 *)
IF Kp_X2 <= 0.0 THEN Kp_X2 := 1.0; END_IF;
IF Ki_X2 <= 0.0 THEN Ki_X2 := 0.1; END_IF;
IF Kd_X2 <= 0.0 THEN Kd_X2 := 0.05; END_IF;

(* Hệ số PID trục Ghép Ms *)
IF Kp_Ms <= 0.0 THEN Kp_Ms := 1.0; END_IF;
IF Ki_Ms <= 0.0 THEN Ki_Ms := 0.1; END_IF;
IF Kd_Ms <= 0.0 THEN Kd_Ms := 0.05; END_IF;

(* Hệ số PID trục Dầu S *)
IF Kp_S <= 0.0 THEN Kp_S := 1.0; END_IF;
IF Ki_S <= 0.0 THEN Ki_S := 0.1; END_IF;
IF Kd_S <= 0.0 THEN Kd_S := 0.05; END_IF;

(* Hệ số PID cuộn Thắng M *)
IF Kp_M <= 0.0 THEN Kp_M := 1.0; END_IF;
IF Ki_M <= 0.0 THEN Ki_M := 0.1; END_IF;
IF Kd_M <= 0.0 THEN Kd_M := 0.05; END_IF;

(* Hệ số PID cuộn Xả U *)
IF Kp_U <= 0.0 THEN Kp_U := 1.0; END_IF;
IF Ki_U <= 0.0 THEN Ki_U := 0.1; END_IF;
IF Kd_U <= 0.0 THEN Kd_U := 0.05; END_IF;

(* ---------------------------------------------------------------------------- *)
(* 9. KHỞI TẠO TORQUE HÃM MIN / MAX VÀ GIỮ DỪNG MÁY (% - REAL)                 *)
(* ---------------------------------------------------------------------------- *)
IF Min_Torque_M          <= 0.0 THEN Min_Torque_M          := 4.0;  END_IF; (* 4.0 % *)
IF Max_Torque_M          <= 0.0 THEN Max_Torque_M          := 20.0; END_IF; (* 20.0 % *)
IF Init_Holding_Torque_M <= 0.0 THEN Init_Holding_Torque_M := 8.0;  END_IF; (* 8.0 % *)

IF Min_Torque_U          <= 0.0 THEN Min_Torque_U          := 5.0;  END_IF; (* 5.0 % *)
IF Max_Torque_U          <= 0.0 THEN Max_Torque_U          := 25.0; END_IF; (* 25.0 % *)
IF Init_Holding_Torque_U <= 0.0 THEN Init_Holding_Torque_U := 10.0; END_IF; (* 10.0 % *)

(* ---------------------------------------------------------------------------- *)
(* 10. KHỞI TẠO HỆ SỐ GAIN CALIB LOADCELL (REAL)                                *)
(* ---------------------------------------------------------------------------- *)
IF Calib_Gain_T  <= 0.0 THEN Calib_Gain_T  := 1.0; END_IF;
IF Calib_Gain_X1 <= 0.0 THEN Calib_Gain_X1 := 1.0; END_IF;
IF Calib_Gain_M  <= 0.0 THEN Calib_Gain_M  := 1.0; END_IF;
IF Calib_Gain_U  <= 0.0 THEN Calib_Gain_U  := 1.0; END_IF;

(* ---------------------------------------------------------------------------- *)
(* 11. KHỞI TẠO CẤU HÌNH MODULE Q68ADV (SLOT 0 - HEAD ADDRESS H00)             *)
(* ---------------------------------------------------------------------------- *)
(* BFM #0: Cho phép chuyển đổi A/D cả 8 kênh (0 = Enable, 1 = Disable)          *)
U0\G0 := 16#0000; (* Enable toàn bộ CH1..CH8 *)

(* BFM #9 & #10: Cài đặt chế độ lọc trung bình trượt (Moving Average = 16#3333) *)
U0\G9  := 16#3333; (* CH1..CH4: Moving Average *)
U0\G10 := 16#3333; (* CH5..CH8: Moving Average *)

(* BFM #11..#18: Số lượng mẫu trung bình trượt (16 mẫu liên tục)                *)
U0\G11 := 16; (* CH1: Loadcell Thu T *)
U0\G12 := 16; (* CH2: Loadcell Kéo X1 *)
U0\G13 := 16; (* CH3: Loadcell Thắng M *)
U0\G14 := 16; (* CH4: Loadcell Xả U *)
U0\G15 := 16; (* CH5: Analog Tốc độ Servo Trục S *)
U0\G16 := 16; (* CH6: Dự phòng *)
U0\G17 := 16; (* CH7: Dự phòng *)
U0\G18 := 16; (* CH8: Dự phòng *)

(* ---------------------------------------------------------------------------- *)
(* 12. KHỞI TẠO CẤU HÌNH MODULE Q68DAV (SLOT 1 - HEAD ADDRESS H10)             *)
(* ---------------------------------------------------------------------------- *)
(* BFM #0: Cho phép chuyển đổi D/A cả 8 kênh (0 = Enable, 1 = Disable)          *)
U1\G0 := 16#0000; (* Enable D/A cho CH1..CH8 *)

(* BFM #9: Cho phép ngõ ra Analog Output (Bit 0..7: 1 = Output Enable)          *)
U1\G9 := 16#00FF; (* Cho phép xuất áp ra cả 8 kênh *)

(* Bật cờ Y11 hoặc Y10 cho phép chuyển đổi D/A *)
Y11 := TRUE;

(* ---- master_all_program.st ---- *)
(* ============================================================================ *)
(* BỘ MÃ NGUỒN GỘP HOÀN CHỈNH TẤT CẢ CHƯƠNG TRÌNH & FUNCTION BLOCK MÁY GHÉP     *)
(* DỰ ÁN: GHEP-MITSU_BACKUP (PLC MITSUBISHI Q02UCPU + CC-LINK)                   *)
(* TÍCH HỢP ĐẦY ĐỦ PHẦN CỨNG THỰC TẾ:                                            *)
(*   1. 5 INPUT SERVO READY (X40..X44) -> NẾU 1 TRỤC NO READY NGẮT DỪNG KHẨN MÁY *)
(*   2. 5 OUTPUT SERVO ON (Y47..Y4B TRÊN QY40)                                  *)
(*   3. CÔNG TẮC GIỮ TORQUE THẮNG M (X45) & XẢ U (X46) CHỐNG TRÙNG MÀNG          *)
(*   4. CÔNG TẮC BÒ CHẬM RỬA MÁY MS (X47) & S (X48) KHI DỪNG MÁY                 *)
(*   5. 2 PEN ÉP MÀNG (Y66, Y67) ĐIỀU KHIỂN TOGGLE (X52, X53) & TỰ NHẢ KHI TỐC CHẬM*)
(*   6. TÍNH ĐƯỜNG KÍNH T THEO ENCODER T & GEAR RATIO T                          *)
(*   7. TÍNH ĐƯỜNG KÍNH M VÀ U THEO 2 CẢM BIẾN TIỆM CẬN X50 & X51                *)
(*   8. NÚT NHẤN VẬT LÝ X49 (START), X4A (STOP), X4B (INC), X4C (DEC)            *)
(*   9. THỜI GIAN GIỮ PHÍM INC/DEC TĂNG/GIẢM TỐC LŨY TIẾN LÊN MAX SPEED         *)
(*  10. CÔN LỰC TAPER TENSION THU T CHỐNG MÓP CUỘN MÀNG                         *)
(* ============================================================================ *)

(******************************************************************************)
(* PHẦN 1: FUNCTION BLOCK 1 - FB_TENSION_PID                                  *)
(* (TẠO TRONG NHÁNH FB/FUN -> ĐẶT TÊN "FB_TENSION_PID")                       *)
(******************************************************************************)

(* --- MÃ ST CHÍNH DÁN VÀO CỬA SỔ FB_TENSION_PID --- *)
IF NOT Enable THEN
    PID_Output := 0;
    I_Term     := 0;
    Error_Prev := 0;
    RETURN;
END_IF;

IF Reset THEN
    I_Term     := 0;
    Error_Prev := 0;
    PID_Output := 0;
    RETURN;
END_IF;

(* 1. Tính độ lệch Error *)
Error := Setpoint - Feedback;

(* 2. Bộ lọc vùng chết Deadband *)
IF ABS(Error) <= Deadband THEN
    Error := 0;
END_IF;

(* 3. Proportional (P) *)
P_Term := (Error * Kp) / 100;

(* 4. Integral (I) có Anti-Windup *)
I_Term := I_Term + ((Error * Ki) / 100);

IF I_Term > Out_Max THEN
    I_Term := Out_Max;
ELSIF I_Term < Out_Min THEN
    I_Term := Out_Min;
END_IF;

(* 5. Derivative (D) *)
D_Term := ((Error - Error_Prev) * Kd) / 100;
Error_Prev := Error;

(* 6. Tổng hợp PID Output *)
PID_Output := P_Term + I_Term + D_Term;

IF PID_Output > Out_Max THEN
    PID_Output := Out_Max;
ELSIF PID_Output < Out_Min THEN
    PID_Output := Out_Min;
END_IF;

(******************************************************************************)
(* PHẦN 2: FUNCTION BLOCK 2 - FFB_METALIZE_CONTROL (FFB_CCLINK_CONTROL)       *)
(* (TẠO TRONG NHÁNH FB/FUN -> ĐẶT TÊN "FFB_CCLINK_CONTROL")                   *)
(******************************************************************************)

(* --- MÃ ST CỦA FFB_CCLINK_CONTROL --- *)
IF Enable THEN
    (* 1. KIỂM TRA TRẠNG THÁI MẠNG CC-LINK (SB0020=0 và SB0049=0 là bình thường) *)
    CCLink_OK := (NOT SB0020) AND (NOT SB0049);
    HasError  := SB0020 OR SB0049 OR M1032 OR M1066;

    M1208 := CCLink_OK;  (* RY8: AD Conversion Enable *)
    M1240 := CCLink_OK;  (* RY28: DA Conversion Enable *)

    (* 2. ĐỌC 4 KÊNH ANALOG INPUT (AJ65SBT-64AD - TRẠM 1) *)
    IF M1016 THEN (* RX8: AD Conversion Completed *)
        ADC_CH1_Raw := D500;
        ADC_CH2_Raw := D501;
        ADC_CH3_Raw := D502;
        ADC_CH4_Raw := D503;

        (* Quy đổi sang 0..1000 (0.0% .. 100.0%) *)
        ADC_CH1_Val := INT_TO_WORD(WORD_TO_INT(D500) * 1000 / 4000);
        ADC_CH2_Val := INT_TO_WORD(WORD_TO_INT(D501) * 1000 / 4000);
        ADC_CH3_Val := INT_TO_WORD(WORD_TO_INT(D502) * 1000 / 4000);
        ADC_CH4_Val := INT_TO_WORD(WORD_TO_INT(D503) * 1000 / 4000);
    END_IF;

    (* 3. GHI 8 KÊNH ANALOG OUTPUT (AJ65VBTCU-68DAVN - TRẠM 2 & 3) *)
    (* QUY ĐỔI LỆNH 0..1000 RA DẢI DAC 0..4000 *)
    D524 := INT_TO_WORD(WORD_TO_INT(Set_Speed_T)  * 4000 / 1000);
    D525 := INT_TO_WORD(WORD_TO_INT(Set_Torque_T) * 4000 / 1000);
    D526 := INT_TO_WORD(WORD_TO_INT(Set_Speed_X1) * 4000 / 1000);
    D527 := INT_TO_WORD(WORD_TO_INT(Set_Speed_X2) * 4000 / 1000);
    D528 := INT_TO_WORD(WORD_TO_INT(Set_Speed_Ms) * 4000 / 1000);
    D529 := INT_TO_WORD(WORD_TO_INT(Set_Torque_M) * 4000 / 1000);
    D530 := INT_TO_WORD(WORD_TO_INT(Set_Speed_S)  * 4000 / 1000);
    D531 := INT_TO_WORD(WORD_TO_INT(Set_Speed_U)  * 4000 / 1000);

    (* 4. XỬ LÝ DIGITAL REMOTE I/O (AJ65SBTB1-16DT: X0..X7 = M1104..M1111 | Y8..YF = M1304..M1311) *)
    DI_X0_State := M1104;
    DI_X1_State := M1105;

    (* Ngõ ra Y8..YF (M1304..M1311) để HMI / User tự set ON/OFF trực tiếp *)

    (* 5. RESET LỖI *)
    M1226 := ResetErr OR M1111; (* RY1A: Reset lỗi trạm 1 *)
    M1258 := ResetErr OR M1111; (* RY3A: Reset lỗi trạm 2 *)
END_IF;

(******************************************************************************)
(* PHẦN 3: PROGRAM CHÍNH - POU_01 (POU_MAIN_METALIZE)                         *)
(* (DÁN VÀO CỬA SỔ POU -> Program -> POU_01)                                   *)
(******************************************************************************)

(* 0. KHỐI KHAI BÁO TỶ SỐ TRUYỀN HỘP SỐ GEAR RATIO ĐỂ RIÊNG ĐỂ DỄ CHỈNH *)
IF Gear_Ratio_T  <= 0 THEN Gear_Ratio_T  := 10100; END_IF; (* Tỷ số truyền 10.1:1 cuộn Thu T *)
IF Gear_Ratio_X1 <= 0 THEN Gear_Ratio_X1 := 8000;  END_IF; (* Tỷ số truyền 8.0:1 kéo X1 *)
IF Gear_Ratio_X2 <= 0 THEN Gear_Ratio_X2 := 8000;  END_IF; (* Tỷ số truyền 8.0:1 Master X2 *)
IF Gear_Ratio_Ms <= 0 THEN Gear_Ratio_Ms := 10000; END_IF; (* Tỷ số truyền 10.0:1 Ghép Ms *)
IF Gear_Ratio_S  <= 0 THEN Gear_Ratio_S  := 10000; END_IF; (* Tỷ số truyền 10.0:1 Dầu S *)
IF Gear_Ratio_U  <= 0 THEN Gear_Ratio_U  := 1000;  END_IF; (* Tỷ số truyền 1.0:1 Xả U *)

(* BẢO VỆ CHỐNG LỖI CHIA CHO 0 & KHỞI TẠO MẶC ĐỊNH *)
IF Max_Speed_MPM <= 0 THEN Max_Speed_MPM := 1000; END_IF;
IF Core_Dia_T_mm <= 0 THEN Core_Dia_T_mm := 76; END_IF;
IF Core_Dia_M_mm <= 0 THEN Core_Dia_M_mm := 76; END_IF;
IF Core_Dia_U_mm <= 0 THEN Core_Dia_U_mm := 76; END_IF;
IF Max_Dia_M_mm  <= 0 THEN Max_Dia_M_mm  := 600; END_IF;
IF Max_Dia_U_mm  <= 0 THEN Max_Dia_U_mm  := 800; END_IF;

IF Speed_Ratio_Ms   <= 0 THEN Speed_Ratio_Ms   := 1000; END_IF; (* Mặc định 100.0% *)
IF Dia_Ms_Roller_mm <= 0 THEN Dia_Ms_Roller_mm := 2000; END_IF; (* Mặc định lô Ms 200.0 mm *)
IF Dia_X2_Roller_mm <= 0 THEN Dia_X2_Roller_mm := 3005; END_IF; (* Mặc định lô X2 300.5 mm *)
IF Decel_Distance_Meters <= 0 THEN Decel_Distance_Meters := 50; END_IF; (* Báo giảm tốc trước 50m *)

IF Ramp_Accel_Rate <= 0 THEN Ramp_Accel_Rate := 5; END_IF;  (* Tăng tốc 5 m/phút mỗi giây *)
IF Ramp_Decel_Rate <= 0 THEN Ramp_Decel_Rate := 10; END_IF; (* Giảm tốc 10 m/phút mỗi giây *)
IF Release_Pen_Speed_MPM <= 0 THEN Release_Pen_Speed_MPM := 20; END_IF; (* 2.0 m/p tự nhả 2 pen *)

(* 1. KIỂM TRA BẢO VỆ 5 TRỤC SERVO READY TRÊN MODULE 16DT (X0..X4 = M1104..M1108) *)
Servo_Not_Ready_Fault := NOT(Servo_Ready_T) OR NOT(Servo_Ready_X1) OR NOT(Servo_Ready_X2) OR NOT(Servo_Ready_Ms) OR NOT(Servo_Ready_S);

IF Servo_Not_Ready_Fault THEN
    State_Machine := 0; (* Ngắt về trạng thái STOPPED khẩn cấp *)
END_IF;

(* 2. ĐIỀU KHIỂN CÔNG TẮC GIỮ TORQUE VÀ CÔNG TẮC BÒ CHẬM RỬA MÁY TRÊN QX40 (X58..X5B) *)
Hold_Torque_Stop_M := Switch_Hold_M;   (* X58 trên QX40 *)
Hold_Torque_Stop_U := Switch_Hold_U;   (* X59 trên QX40 *)
Anti_Dry_Rotate_Ms := Switch_Wash_Ms;  (* X5A trên QX40 *)
Anti_Dry_Rotate_S  := Switch_Wash_S;   (* X5B trên QX40 *)

(* 3. NẠP LẠI ĐƯỜNG KÍNH KHI NẠP CUỘN MỚI *)
IF HMI_Reset_Roll_T THEN Real_Dia_T_mm := Core_Dia_T_mm; HMI_Reset_Roll_T := FALSE; END_IF;
IF HMI_Reset_Roll_M THEN Real_Dia_M_mm := Max_Dia_M_mm;  HMI_Reset_Roll_M := FALSE; END_IF;
IF HMI_Reset_Roll_U THEN Real_Dia_U_mm := Max_Dia_U_mm;  HMI_Reset_Roll_U := FALSE; END_IF;

(* 4. TỔNG HỢP NÚT NHẤN HMI & NÚT NHẤN VẬT LÝ (X49, X4A, X4B, X4C) *)
Cmd_Start := HMI_Start OR Physical_Start_PB;
Cmd_Stop  := HMI_Stop OR Physical_Stop_PB OR Servo_Not_Ready_Fault;
Cmd_Inc   := HMI_Inc_Hold OR Physical_Inc_PB;
Cmd_Dec   := HMI_Dec_Hold OR Physical_Dec_PB;

(* 5. ĐIỀU KHIỂN TOGGLE 2 PEN ÉP MÀNG (Y66, Y67) & TỰ NHẢ KHI TỐC CHẬM *)
Trig_Pen1 := (Pen1_Toggle_PB AND NOT(Prev_Pen1_PB)) OR HMI_Pen1_Cmd;
Prev_Pen1_PB := Pen1_Toggle_PB;
IF HMI_Pen1_Cmd THEN HMI_Pen1_Cmd := FALSE; END_IF;
IF Trig_Pen1 THEN Pen1_State := NOT(Pen1_State); END_IF;

Trig_Pen2 := (Pen2_Toggle_PB AND NOT(Prev_Pen2_PB)) OR HMI_Pen2_Cmd;
Prev_Pen2_PB := Pen2_Toggle_PB;
IF HMI_Pen2_Cmd THEN HMI_Pen2_Cmd := FALSE; END_IF;
IF Trig_Pen2 THEN Pen2_State := NOT(Pen2_State); END_IF;

(* TỰ ĐỘNG NHẢ 2 PEN KHI MÁY GIẢM VỀ TỐC ĐỘ CHẬM HOẶC DỪNG MÁY *)
IF Current_Line_MPM <= Release_Pen_Speed_MPM OR State_Machine = 0 THEN
    Pen1_State := FALSE;
    Pen2_State := FALSE;
END_IF;

(* XUẤT 2 ĐẦU RA PEN ÉP MÀNG RA MODULE 16DT CC-LINK (YD=M1309, YE=M1310) *)
M1309 := Pen1_State; (* Ngõ ra Pen 1 -> Cọc YD (Cọc 6) trên Module 16DT *)
M1310 := Pen2_State; (* Ngõ ra Pen 2 -> Cọc YE (Cọc 7) trên Module 16DT *)

(* 6. TĂNG GIẢM TỐC LŨY TIẾN THEO THỜI GIAN GIỮ PHÍM INC / DEC *)
IF Cmd_Inc THEN
    Inc_Hold_Timer := Inc_Hold_Timer + 1;
    IF Inc_Hold_Timer < 50 THEN
        Dynamic_Accel_Step := Ramp_Accel_Rate;
    ELSIF Inc_Hold_Timer < 150 THEN
        Dynamic_Accel_Step := Ramp_Accel_Rate * 2;
    ELSE
        Dynamic_Accel_Step := Ramp_Accel_Rate * 5; (* Bấm giữ lâu tăng tốc vọt lên *)
    END_IF;
    Target_Line_MPM := Target_Line_MPM + Dynamic_Accel_Step;
    IF Target_Line_MPM > Max_Speed_MPM THEN Target_Line_MPM := Max_Speed_MPM; END_IF;
ELSE
    Inc_Hold_Timer := 0;
END_IF;

IF Cmd_Dec THEN
    Dec_Hold_Timer := Dec_Hold_Timer + 1;
    IF Dec_Hold_Timer < 50 THEN
        Dynamic_Accel_Step := Ramp_Decel_Rate;
    ELSIF Dec_Hold_Timer < 150 THEN
        Dynamic_Accel_Step := Ramp_Decel_Rate * 2;
    ELSE
        Dynamic_Accel_Step := Ramp_Decel_Rate * 5; (* Bấm giữ lâu giảm tốc vọt xuống *)
    END_IF;
    Target_Line_MPM := Target_Line_MPM - Dynamic_Accel_Step;
    IF Target_Line_MPM < Min_Speed_MPM THEN Target_Line_MPM := Min_Speed_MPM; END_IF;
ELSE
    Dec_Hold_Timer := 0;
END_IF;

(* Ramping tốc độ hiện tại tiến dần đến tốc độ mục tiêu *)
IF Current_Line_MPM < Target_Line_MPM THEN
    Current_Line_MPM := Current_Line_MPM + Ramp_Accel_Rate;
    IF Current_Line_MPM > Target_Line_MPM THEN Current_Line_MPM := Target_Line_MPM; END_IF;
ELSIF Current_Line_MPM > Target_Line_MPM THEN
    Current_Line_MPM := Current_Line_MPM - Ramp_Decel_Rate;
    IF Current_Line_MPM < Target_Line_MPM THEN Current_Line_MPM := Target_Line_MPM; END_IF;
END_IF;

(* 7. TÍNH ĐƯỜNG KÍNH THỰC TẾ 3 CUỘN T, M, U *)
(* --- 7A. Tính đường kính cuộn Thu T theo Encoder T & Gear_Ratio_T --- *)
Curr_Pulse_T  := INT_TO_DINT(D5000); (* Đọc từ High-speed Counter QD62 Module *)
Curr_Pulse_X2 := INT_TO_DINT(D5002); (* Đọc xung Master X2 Encoder *)

IF (Curr_Pulse_T - Last_Pulse_T) >= ((8000 * Gear_Ratio_T) / 1000) THEN
    Rev_Count_T := Rev_Count_T + 1;
    IF (Curr_Pulse_X2 - Last_Pulse_X2_T) > 0 THEN
        Raw_Dia_T_mm := ((Curr_Pulse_X2 - Last_Pulse_X2_T) * Dia_X2_Roller_mm) / 320000;
        IF Raw_Dia_T_mm < Core_Dia_T_mm THEN Raw_Dia_T_mm := Core_Dia_T_mm; END_IF;
        IF Raw_Dia_T_mm > Max_Dia_T_mm THEN Raw_Dia_T_mm := Max_Dia_T_mm; END_IF;
        Real_Dia_T_mm := Real_Dia_T_mm + ((Raw_Dia_T_mm - Real_Dia_T_mm) / 5);
    END_IF;
    Last_Pulse_X2_T := Curr_Pulse_X2;
    Last_Pulse_T    := Curr_Pulse_T;
END_IF;

(* --- 7B. Tính đường kính cuộn M theo cảm biến tiệm cận X50 --- *)
Trig_X50 := Sensor_Rev_M AND NOT(Prev_X50);
Prev_X50 := Sensor_Rev_M;

IF Trig_X50 THEN
    Rev_Count_M := Rev_Count_M + 1;
    IF (Curr_Pulse_X2 - Last_Pulse_X2_M) > 0 THEN
        Raw_Dia_M_mm := ((Curr_Pulse_X2 - Last_Pulse_X2_M) * Dia_X2_Roller_mm) / 320000;
        IF Raw_Dia_M_mm < Core_Dia_M_mm THEN Raw_Dia_M_mm := Core_Dia_M_mm; END_IF;
        IF Raw_Dia_M_mm > Max_Dia_M_mm THEN Raw_Dia_M_mm := Max_Dia_M_mm; END_IF;
        Real_Dia_M_mm := Real_Dia_M_mm + ((Raw_Dia_M_mm - Real_Dia_M_mm) / 5);
    END_IF;
    Last_Pulse_X2_M := Curr_Pulse_X2;
END_IF;

(* --- 7C. Tính đường kính cuộn U theo cảm biến tiệm cận X51 --- *)
Trig_X51 := Sensor_Rev_U AND NOT(Prev_X51);
Prev_X51 := Sensor_Rev_U;

IF Trig_X51 THEN
    Rev_Count_U := Rev_Count_U + 1;
    IF (Curr_Pulse_X2 - Last_Pulse_X2_U) > 0 THEN
        Raw_Dia_U_mm := ((Curr_Pulse_X2 - Last_Pulse_X2_U) * Dia_X2_Roller_mm) / 320000;
        IF Raw_Dia_U_mm < Core_Dia_U_mm THEN Raw_Dia_U_mm := Core_Dia_U_mm; END_IF;
        IF Raw_Dia_U_mm > Max_Dia_U_mm THEN Raw_Dia_U_mm := Max_Dia_U_mm; END_IF;
        Real_Dia_U_mm := Real_Dia_U_mm + ((Raw_Dia_U_mm - Real_Dia_U_mm) / 5);
    END_IF;
    Last_Pulse_X2_U := Curr_Pulse_X2;
END_IF;

(* 8. STATE MACHINE VẬN HÀNH DÂY CHUYỀN *)
CASE State_Machine OF
    0: (* STATE_STOPPED *)
        Current_Line_MPM := 0;
        Target_Line_MPM  := 0;

        IF Cmd_Start AND NOT(Servo_Not_Ready_Fault) THEN
            State_Machine := 1;
            HMI_Start := FALSE;
        END_IF;

    1: (* STATE_RUNNING *)
        IF Cmd_Stop THEN
            State_Machine := 0;
            HMI_Stop := FALSE;
        END_IF;
END_CASE;

(* TẬP TRUNG TÍN HIỆU 5 TRỤC SERVO ON XUẤT RA MODULE 16DT CC-LINK (Y8..YC = M1304..M1308) *)
M1304 := (State_Machine = 1);                                                (* Y8 (Cọc 1): Servo ON Thu T *)
M1305 := (State_Machine = 1);                                                (* Y9 (Cọc 2): Servo ON Xả X1 *)
M1306 := (State_Machine = 1);                                                (* YA (Cọc 3): Servo ON Master X2 *)
M1307 := (State_Machine = 1) OR (State_Machine = 0 AND Anti_Dry_Rotate_Ms);  (* YB (Cọc 4): Servo ON Ghép Ms *)
M1308 := (State_Machine = 1) OR (State_Machine = 0 AND Anti_Dry_Rotate_S);   (* YC (Cọc 5): Servo ON Tráng Dầu S *)

Servo_ON_T  := M1304;
Servo_ON_X1 := M1305;
Servo_ON_X2 := M1306;
Servo_ON_Ms := M1307;
Servo_ON_S  := M1308;

(* 9. TÍNH CÔN LỰC TAPER TENSION CHO CUỘN THU T *)
IF (Max_Dia_T_mm - Core_Dia_T_mm) > 0 AND Taper_Percent_T > 0 THEN
    Effective_SP_T := SP_Tension_T - (((Real_Dia_T_mm - Core_Dia_T_mm) * SP_Tension_T * Taper_Percent_T) / ((Max_Dia_T_mm - Core_Dia_T_mm) * 100));
ELSE
    Effective_SP_T := SP_Tension_T;
END_IF;

IF Effective_SP_T < 0 THEN Effective_SP_T := 0; END_IF;

(* TẠO XUNG KÍCH HOẠT PID CHUẨN 10MS TỪ SM409 (0.01s CLOCK) *)
Trig_PID_10ms := SM409 AND NOT(Prev_SM409);
Prev_SM409 := SM409;

(* 10. GỌI RUN 4 INSTANCE PID MỖI CHU KỲ 10MS ĐỂ TRÁNH TRÔI TÍCH PHÂN & BẢO ĐẢM TỐC ĐỘ QUÉT X50/X51 *)
IF Trig_PID_10ms THEN
    pid_T(Enable := HMI_PID_Enable, Setpoint := Effective_SP_T, Feedback := Weight_Net_T, Kp := Kp_T, Ki := Ki_T, Kd := Kd_T);
    pid_X1(Enable := HMI_PID_Enable, Setpoint := SP_Tension_X1, Feedback := Weight_Net_X1, Kp := Kp_X1, Ki := Ki_X1, Kd := Kd_X1);
    pid_M(Enable := HMI_PID_Enable, Setpoint := SP_Tension_M, Feedback := Weight_Net_M, Kp := Kp_M, Ki := Ki_M, Kd := Kd_M);
    pid_U(Enable := HMI_PID_Enable, Setpoint := SP_Tension_U, Feedback := Weight_Net_U, Kp := Kp_U, Ki := Ki_U, Kd := Kd_U);

    PID_Out_T  := pid_T.PID_Output;
    PID_Out_X1 := pid_X1.PID_Output;
    PID_Out_M  := pid_M.PID_Output;
    PID_Out_U  := pid_U.PID_Output;
END_IF;

(* 11. TÍNH TOÁN CÁC GIÁ TRỊ TỐC ĐỘ VÀ TORQUE TỪ BIẾN LOCAL PID *)
IF State_Machine = 0 THEN
    Calc_Speed_T  := 0;
    Calc_Speed_X1 := 0;

    IF Anti_Dry_Rotate_Ms THEN
        Calc_Speed_Ms := (Anti_Dry_Crawl_Speed * 4000) / Max_Speed_MPM;
    ELSE
        Calc_Speed_Ms := 0;
    END_IF;

    IF Anti_Dry_Rotate_S THEN
        Calc_Speed_S := (Anti_Dry_Crawl_Speed * 4000) / Max_Speed_MPM;
    ELSE
        Calc_Speed_S := 0;
    END_IF;

    IF Hold_Torque_Stop_M THEN
        Calc_Torque_M := Base_Torque_M;
    ELSE
        Calc_Torque_M := 0;
    END_IF;

    IF Hold_Torque_Stop_U THEN
        Calc_Speed_U := Init_Holding_Torque_U;
    ELSE
        Calc_Speed_U := 0;
    END_IF;
ELSE
    (* CHẠY TỰ ĐỘNG *)
    IF Dia_X2_Roller_mm > 0 THEN
        Calc_Speed_Ms := (((Calc_Speed_X2 * Dia_Ms_Roller_mm) / Dia_X2_Roller_mm) * Speed_Ratio_Ms) / 1000;
    ELSE
        Calc_Speed_Ms := Calc_Speed_X2;
    END_IF;

    IF Real_Dia_T_mm > 0 THEN
        Calc_Speed_T := ((Calc_Speed_X2 * Real_Dia_T_mm) / Core_Dia_T_mm) + PID_Out_T;
    ELSE
        Calc_Speed_T := Calc_Speed_X2 + PID_Out_T;
    END_IF;

    Calc_Speed_X1 := Calc_Speed_X2 + PID_Out_X1;
    Calc_Speed_S  := ((Calc_Speed_X2 * Speed_Ratio_S) / 1000) + Speed_Offset_S;
    IF Calc_Speed_S < 0 THEN Calc_Speed_S := 0; END_IF;
    IF Calc_Speed_S > 4000 THEN Calc_Speed_S := 4000; END_IF;

    IF Real_Dia_U_mm > 0 THEN
        Calc_Speed_U := ((Calc_Speed_X2 * Max_Dia_U_mm) / Real_Dia_U_mm) + PID_Out_U;
    ELSE
        Calc_Speed_U := Calc_Speed_X2 + PID_Out_U;
    END_IF;

    Calc_Torque_M := Base_Torque_M + PID_Out_M;
END_IF;

(* 12. Thực thi FB CC-Link Master với Ép kiểu DINT_TO_WORD *)
fbCCLink(
    Enable          := TRUE,
    ResetErr        := HMI_Reset_Error,
    Auto_Mode       := HMI_Auto_Mode,
    Set_Speed_T     := DINT_TO_WORD(Calc_Speed_T),
    Set_Torque_T    := DINT_TO_WORD(PID_Out_T),
    Set_Speed_X1    := DINT_TO_WORD(Calc_Speed_X1),
    Set_Speed_X2    := DINT_TO_WORD(Calc_Speed_X2),
    Set_Speed_Ms    := DINT_TO_WORD(Calc_Speed_Ms),
    Set_Torque_M    := DINT_TO_WORD(Calc_Torque_M),
    Set_Speed_S     := DINT_TO_WORD(Calc_Speed_S),
    Set_Speed_U     := DINT_TO_WORD(Calc_Speed_U)
);

(* 13. TỰ ĐỘNG BÁO GIẢM TỐC KHI GẦN ĐẠT CHIỀU DÀI MÉT CÀI ĐẶT *)
IF Set_Target_Length > 0 AND Decel_Distance_Meters > 0 THEN
    IF Total_Length_Meters >= (Set_Target_Length - Decel_Distance_Meters) THEN
        Auto_Decel_Flag := TRUE;
        IF Target_Line_MPM > Min_Speed_MPM THEN Target_Line_MPM := Min_Speed_MPM; END_IF;
    ELSE
        Auto_Decel_Flag := FALSE;
    END_IF;
END_IF;

(* 14. TÍNH TỐC ĐỘ MASTER X2 *)
Calc_Speed_X2 := (Current_Line_MPM * 4000) / Max_Speed_MPM;

(* ---- metalize_cclink_fb.st ---- *)
(* ============================================================================ *)
(* FUNCTION BLOCK: FFB_METALIZE_CONTROL                                         *)
(* DỰ ÁN: QUẢN LÝ DÂY CHUYỀN MÁY GHÉP MÀNG METALIZE (Q02U + CC-LINK)            *)
(* PHẦN CỨNG:                                                                   *)
(*   - Trạm 1 (AJ65SBT-64AD): 4 CH Loadcell (Zero & Calib Gain)                 *)
(*   - Trạm 2&3 (AJ65VBTCU-68DAVN): 8 CH DAC Output (Ramping Tăng/Giảm Tốc)     *)
(*   - Trạm 4 (AJ65SBT-16DT): 5 Trục Servo Ready & Servo ON                     *)
(* ============================================================================ *)

VAR_INPUT
    Enable          : BOOL := TRUE;  (* Cho phep FB hoat dong *)
    ResetErr        : BOOL := FALSE; (* Nut Reset loi he thong *)
    Auto_Mode       : BOOL := TRUE;  (* TRUE: Tu dong, FALSE: Manual Test *)

    (* LỆNH SET ZERO VÀ HỆ SỐ CALIB LOADCELL (4 CH TRẠM 1) *)
    Zero_Set_T      : BOOL := FALSE;
    Zero_Set_X1     : BOOL := FALSE;
    Zero_Set_M      : BOOL := FALSE;
    Zero_Set_U      : BOOL := FALSE;

    Calib_Gain_T    : DINT := 1000;
    Calib_Gain_X1   : DINT := 1000;
    Calib_Gain_M    : DINT := 1000;
    Calib_Gain_U    : DINT := 1000;

    (* CÀI ĐẶT TỐC ĐỘ VÀ TORQUE TỪ CHƯƠNG TRÌNH CHÍNH (0..4000) *)
    Set_Speed_T     : WORD := 0; (* CH1: Speed Thu T *)
    Set_Torque_T    : WORD := 0; (* CH2: Torque Thu T *)
    Set_Speed_X1    : WORD := 0; (* CH3: Speed Xa Giay X1 *)
    Set_Speed_X2    : WORD := 0; (* CH4: Speed Master X2 *)
    Set_Speed_Ms    : WORD := 0; (* CH5: Speed Ghep Metalize Ms *)
    Set_Torque_M    : WORD := 0; (* CH6: Torque Thang Tu M *)
    Set_Speed_S     : WORD := 0; (* CH7: Speed Trang Dau S *)
    Set_Speed_U     : WORD := 0; (* CH8: Speed Xa Metalize U *)

    (* BƯỚC TĂNG GIẢM TỐC RAMPING *)
    Ramp_Step_ms    : DINT := 20;

    (* LỆNH SERVO ON CHẾ ĐỘ TỰ ĐỘNG *)
    Auto_Son_T      : BOOL := FALSE;
    Auto_Son_X1     : BOOL := FALSE;
    Auto_Son_X2     : BOOL := FALSE;
    Auto_Son_M      : BOOL := FALSE;
    Auto_Son_S      : BOOL := FALSE;

    (* LỆNH TEST TỪNG TRỤC CHẾ ĐỘ MANUAL *)
    Test_Son_T      : BOOL := FALSE;
    Test_Son_X1     : BOOL := FALSE;
    Test_Son_X2     : BOOL := FALSE;
    Test_Son_M      : BOOL := FALSE;
    Test_Son_S      : BOOL := FALSE;

    Test_Speed_T    : WORD := 0;
    Test_Speed_X1   : WORD := 0;
    Test_Speed_X2   : WORD := 0;
    Test_Speed_Ms   : WORD := 0;
    Test_Torque_M   : WORD := 0;
    Test_Speed_S    : WORD := 0;
    Test_Speed_U    : WORD := 0;
END_VAR

VAR_OUTPUT
    CCLink_OK       : BOOL := FALSE; (* Bao truyen thong CC-Link OK *)
    HasError        : BOOL := FALSE; (* Bao loi he thong *)

    (* GIÁ TRỊ TRỌNG LƯỢNG / LỰC CĂNG NET SAU CALIB & ZERO (0..4000 N/Kg) *)
    Weight_Net_T    : DINT := 0; (* CH1 *)
    Weight_Net_X1   : DINT := 0; (* CH2 *)
    Weight_Net_M    : DINT := 0; (* CH3 *)
    Weight_Net_U    : DINT := 0; (* CH4 *)

    (* TRẠNG THÁI SERVO READY VÀ SERVO ON *)
    S_Ready_T       : BOOL := FALSE;
    S_Ready_X1      : BOOL := FALSE;
    S_Ready_X2      : BOOL := FALSE;
    S_Ready_M       : BOOL := FALSE;
    S_Ready_S       : BOOL := FALSE;

    S_ON_T_Out      : BOOL := FALSE;
    S_ON_X1_Out     : BOOL := FALSE;
    S_ON_X2_Out     : BOOL := FALSE;
    S_ON_M_Out      : BOOL := FALSE;
    S_ON_S_Out      : BOOL := FALSE;
END_VAR

VAR
    Zero_Offset_T   : DINT := 0;
    Zero_Offset_X1  : DINT := 0;
    Zero_Offset_M   : DINT := 0;
    Zero_Offset_U   : DINT := 0;

    Ramp_Speed_T    : DINT := 0;
    Ramp_Torque_T   : DINT := 0;
    Ramp_Speed_X1   : DINT := 0;
    Ramp_Speed_X2   : DINT := 0;
    Ramp_Speed_Ms   : DINT := 0;
    Ramp_Torque_M   : DINT := 0;
    Ramp_Speed_S    : DINT := 0;
    Ramp_Speed_U    : DINT := 0;

    Target_D524     : DINT := 0;
    Target_D525     : DINT := 0;
    Target_D526     : DINT := 0;
    Target_D527     : DINT := 0;
    Target_D528     : DINT := 0;
    Target_D529     : DINT := 0;
    Target_D530     : DINT := 0;
    Target_D531     : DINT := 0;
END_VAR

IF Enable THEN

    (* 1. KIỂM TRA MẠNG CC-LINK *)
    CCLink_OK := SB0020;
    HasError  := NOT(SB0020) OR M1032 OR M1066;

    M1208 := SB0020; (* RY8: Kick ADC Tram 1 *)
    M1240 := SB0020; (* RY28: Kick DAC Tram 2 *)

    (* 2. ĐỌC VÀ HIỆU CHUẨN (CALIB & ZERO) 4 KÊNH LOADCELL (TRẠM 1 - AJ65SBT-64AD) *)
    IF M1016 THEN (* RX8 *)
        IF Zero_Set_T  THEN Zero_Offset_T  := WORD_TO_INT(D500); END_IF;
        IF Zero_Set_X1 THEN Zero_Offset_X1 := WORD_TO_INT(D501); END_IF;
        IF Zero_Set_M  THEN Zero_Offset_M  := WORD_TO_INT(D502); END_IF;
        IF Zero_Set_U  THEN Zero_Offset_U  := WORD_TO_INT(D503); END_IF;

        Weight_Net_T  := ((WORD_TO_INT(D500) - Zero_Offset_T)  * Calib_Gain_T)  / 1000;
        Weight_Net_X1 := ((WORD_TO_INT(D501) - Zero_Offset_X1) * Calib_Gain_X1) / 1000;
        Weight_Net_M  := ((WORD_TO_INT(D502) - Zero_Offset_M)  * Calib_Gain_M)  / 1000;
        Weight_Net_U  := ((WORD_TO_INT(D503) - Zero_Offset_U)  * Calib_Gain_U)  / 1000;

        IF Weight_Net_T  < 0 THEN Weight_Net_T  := 0; END_IF;
        IF Weight_Net_X1 < 0 THEN Weight_Net_X1 := 0; END_IF;
        IF Weight_Net_M  < 0 THEN Weight_Net_M  := 0; END_IF;
        IF Weight_Net_U  < 0 THEN Weight_Net_U  := 0; END_IF;
    END_IF;

    (* 3. LỰA CHỌN MỤC TIÊU TỐC ĐỘ VÀ RAMPING TĂNG GIẢM TỐC *)
    IF Auto_Mode THEN
        Target_D524 := WORD_TO_INT(Set_Speed_T)  / 2;
        Target_D525 := WORD_TO_INT(Set_Torque_T) / 2;
        Target_D526 := WORD_TO_INT(Set_Speed_X1) / 2;
        Target_D527 := WORD_TO_INT(Set_Speed_X2) / 2;
        Target_D528 := WORD_TO_INT(Set_Speed_Ms) / 2;
        Target_D529 := WORD_TO_INT(Set_Torque_M) / 2;
        Target_D530 := WORD_TO_INT(Set_Speed_S)  / 2;
        Target_D531 := WORD_TO_INT(Set_Speed_U)  / 2;

        S_ON_T_Out  := Auto_Son_T  AND SB0020;
        S_ON_X1_Out := Auto_Son_X1 AND SB0020;
        S_ON_X2_Out := Auto_Son_X2 AND SB0020;
        S_ON_M_Out  := Auto_Son_M  AND SB0020;
        S_ON_S_Out  := Auto_Son_S  AND SB0020;
    ELSE
        Target_D524 := WORD_TO_INT(Test_Speed_T)  / 2;
        Target_D525 := 0;
        Target_D526 := WORD_TO_INT(Test_Speed_X1) / 2;
        Target_D527 := WORD_TO_INT(Test_Speed_X2) / 2;
        Target_D528 := WORD_TO_INT(Test_Speed_Ms) / 2;
        Target_D529 := WORD_TO_INT(Test_Torque_M) / 2;
        Target_D530 := WORD_TO_INT(Test_Speed_S)  / 2;
        Target_D531 := WORD_TO_INT(Test_Speed_U)  / 2;

        S_ON_T_Out  := Test_Son_T  AND SB0020;
        S_ON_X1_Out := Test_Son_X1 AND SB0020;
        S_ON_X2_Out := Test_Son_X2 AND SB0020;
        S_ON_M_Out  := Test_Son_M  AND SB0020;
        S_ON_S_Out  := Test_Son_S  AND SB0020;
    END_IF;

    (* RAMPING TĂNG GIẢM TỐC CHỐNG ĐỨT MÀNG (ACCEL/DECEL RAMP) *)
    IF Ramp_Speed_T < Target_D524 THEN Ramp_Speed_T := Ramp_Speed_T + Ramp_Step_ms; IF Ramp_Speed_T > Target_D524 THEN Ramp_Speed_T := Target_D524; END_IF;
    ELSIF Ramp_Speed_T > Target_D524 THEN Ramp_Speed_T := Ramp_Speed_T - Ramp_Step_ms; IF Ramp_Speed_T < Target_D524 THEN Ramp_Speed_T := Target_D524; END_IF; END_IF;

    IF Ramp_Speed_X1 < Target_D526 THEN Ramp_Speed_X1 := Ramp_Speed_X1 + Ramp_Step_ms; IF Ramp_Speed_X1 > Target_D526 THEN Ramp_Speed_X1 := Target_D526; END_IF;
    ELSIF Ramp_Speed_X1 > Target_D526 THEN Ramp_Speed_X1 := Ramp_Speed_X1 - Ramp_Step_ms; IF Ramp_Speed_X1 < Target_D526 THEN Ramp_Speed_X1 := Target_D526; END_IF; END_IF;

    IF Ramp_Speed_X2 < Target_D527 THEN Ramp_Speed_X2 := Ramp_Speed_X2 + Ramp_Step_ms; IF Ramp_Speed_X2 > Target_D527 THEN Ramp_Speed_X2 := Target_D527; END_IF;
    ELSIF Ramp_Speed_X2 > Target_D527 THEN Ramp_Speed_X2 := Ramp_Speed_X2 - Ramp_Step_ms; IF Ramp_Speed_X2 < Target_D527 THEN Ramp_Speed_X2 := Target_D527; END_IF; END_IF;

    IF Ramp_Speed_Ms < Target_D528 THEN Ramp_Speed_Ms := Ramp_Speed_Ms + Ramp_Step_ms; IF Ramp_Speed_Ms > Target_D528 THEN Ramp_Speed_Ms := Target_D528; END_IF;
    ELSIF Ramp_Speed_Ms > Target_D528 THEN Ramp_Speed_Ms := Ramp_Speed_Ms - Ramp_Step_ms; IF Ramp_Speed_Ms < Target_D528 THEN Ramp_Speed_Ms := Target_D528; END_IF; END_IF;

    IF Ramp_Speed_S < Target_D530 THEN Ramp_Speed_S := Ramp_Speed_S + Ramp_Step_ms; IF Ramp_Speed_S > Target_D530 THEN Ramp_Speed_S := Target_D530; END_IF;
    ELSIF Ramp_Speed_S > Target_D530 THEN Ramp_Speed_S := Ramp_Speed_S - Ramp_Step_ms; IF Ramp_Speed_S < Target_D530 THEN Ramp_Speed_S := Target_D530; END_IF; END_IF;

    IF Ramp_Speed_U < Target_D531 THEN Ramp_Speed_U := Ramp_Speed_U + Ramp_Step_ms; IF Ramp_Speed_U > Target_D531 THEN Ramp_Speed_U := Target_D531; END_IF;
    ELSIF Ramp_Speed_U > Target_D531 THEN Ramp_Speed_U := Ramp_Speed_U - Ramp_Step_ms; IF Ramp_Speed_U < Target_D531 THEN Ramp_Speed_U := Target_D531; END_IF; END_IF;

    Ramp_Torque_T := Target_D525;
    Ramp_Torque_M := Target_D529;

    D524 := INT_TO_WORD(Ramp_Speed_T);
    D525 := INT_TO_WORD(Ramp_Torque_T);
    D526 := INT_TO_WORD(Ramp_Speed_X1);
    D527 := INT_TO_WORD(Ramp_Speed_X2);
    D528 := INT_TO_WORD(Ramp_Speed_Ms);
    D529 := INT_TO_WORD(Ramp_Torque_M);
    D530 := INT_TO_WORD(Ramp_Speed_S);
    D531 := INT_TO_WORD(Ramp_Speed_U);

    (* 4. ĐỌC SERVO READY VÀ XUẤT SERVO ON (AJ65SBT-16DT - TRẠM 4) *)
    S_Ready_T  := M1104;
    S_Ready_X1 := M1105;
    S_Ready_X2 := M1106;
    S_Ready_M  := M1107;
    S_Ready_S  := M1108;

    M1296 := S_ON_T_Out;
    M1297 := S_ON_X1_Out;
    M1298 := S_ON_X2_Out;
    M1299 := S_ON_M_Out;
    M1300 := S_ON_S_Out;

    M1303 := HasError;

    (* 5. RESET LỖI CC-LINK *)
    M1226 := ResetErr OR M1111;
    M1258 := ResetErr OR M1111;

END_IF;
